C05370=1007.912,298.637,-156.011,2.906,71.013,33.161
C05371=1007.852,298.815,-156.123,3.500,71.107,33.963
C05372=1007.792,298.994,-156.236,4.100,71.198,34.771
C05373=1007.731,299.173,-156.349,4.700,71.282,35.586
C05374=1007.670,299.350,-156.464,5.320,71.368,36.417
C05375=1007.609,299.529,-156.578,5.950,71.452,37.259
C05376=1007.547,299.705,-156.694,6.591,71.533,38.113
C05377=1007.484,299.883,-156.809,7.249,71.615,38.983
C05378=1007.421,300.059,-156.927,7.912,71.693,39.860
C05379=1007.359,300.235,-157.044,8.587,71.769,40.749
C05380=1007.294,300.411,-157.161,9.296,71.851,41.666
C05381=1007.230,300.586,-157.281,9.991,71.920,42.578
C05382=1007.164,300.761,-157.400,10.723,71.997,43.519
C05383=1007.099,300.936,-157.520,11.439,72.060,44.454
C05384=1007.034,301.109,-157.640,12.197,72.133,45.420
C05385=1006.967,301.283,-157.761,12.947,72.195,46.385
C05386=1006.900,301.456,-157.883,13.707,72.254,47.361
C05387=1006.832,301.629,-158.007,14.495,72.315,48.362
C05388=1006.764,301.802,-158.130,15.272,72.365,49.358
C05389=1006.696,301.973,-158.254,16.077,72.419,50.376
C05390=1006.628,302.145,-158.378,16.906,72.473,51.414
C05391=1006.558,302.316,-158.504,17.740,72.521,52.461
C05392=1006.488,302.487,-158.630,18.568,72.561,53.505
C05393=1006.418,302.657,-158.757,19.417,72.600,54.567
C05394=1006.347,302.827,-158.884,20.271,72.636,55.634
C05395=1006.276,302.996,-159.013,21.134,72.666,56.711
C05396=1006.204,303.164,-159.141,22.013,72.694,57.803
C05397=1006.131,303.333,-159.270,22.899,72.718,58.901
C05398=1006.058,303.500,-159.401,23.787,72.735,60.004
C05399=1005.985,303.668,-159.531,24.716,72.757,61.138
C05400=1005.911,303.835,-159.663,25.614,72.764,62.252
C05401=1005.836,304.001,-159.795,26.558,72.775,63.401
C05402=1005.761,304.166,-159.928,27.467,72.773,64.528
C05403=1005.686,304.332,-160.061,28.426,72.776,65.689
C05404=1005.610,304.497,-160.195,29.363,72.767,66.839
C05405=1005.533,304.661,-160.330,30.303,72.753,67.991
C05406=1005.456,304.824,-160.466,31.260,72.738,69.154
C05407=1005.379,304.988,-160.602,32.197,72.712,70.305
C05408=1005.300,305.150,-160.740,33.155,72.686,71.469
C05409=1005.221,305.312,-160.876,34.138,72.658,72.651
C05410=1005.141,305.474,-161.015,35.102,72.622,73.820
C05411=1005.062,305.634,-161.154,36.053,72.578,74.978
C05412=1004.982,305.795,-161.294,37.021,72.531,76.150
C05413=1004.901,305.954,-161.434,37.983,72.478,77.315
C05414=1004.820,306.114,-161.576,38.940,72.419,78.476
C05415=1004.738,306.273,-161.717,39.900,72.356,79.638
C05416=1004.656,306.430,-161.859,40.856,72.287,80.795
C05417=1004.574,306.588,-162.002,41.803,72.212,81.945
C05418=1004.490,306.745,-162.146,42.786,72.137,83.118
C05419=1004.406,306.901,-162.290,43.707,72.048,84.246
C05420=1004.321,307.056,-162.435,44.673,71.960,85.405
C05421=1004.237,307.211,-162.581,45.601,71.862,86.534
C05422=1004.152,307.366,-162.728,46.537,71.762,87.663
C05423=1004.065,307.519,-162.875,47.480,71.659,88.795
C05424=1003.979,307.673,-163.023,48.398,71.548,89.905
C05425=1003.893,307.825,-163.171,49.292,71.430,90.995
C05426=1003.804,307.977,-163.320,50.204,71.310,92.094
C05427=1003.717,308.128,-163.469,51.076,71.182,93.162
C05428=1003.628,308.279,-163.620,51.950,71.050,94.225
C05429=1003.539,308.429,-163.771,52.856,70.919,95.305
C05430=1003.403,308.655,-164.001,54.168,70.704,96.898
C05431=1003.266,308.880,-164.234,55.443,70.477,98.453
C05432=1003.564,308.723,-164.621,36.254,67.418,86.861
C05433=1003.709,308.486,-164.376,34.721,67.533,84.964
C05434=1003.852,308.248,-164.134,33.173,67.628,83.052
C05435=1003.941,308.099,-163.985,32.181,67.673,81.840
C05436=1004.029,307.948,-163.834,31.222,67.719,80.647
C05437=1004.116,307.798,-163.684,30.275,67.761,79.460
C05438=1004.203,307.646,-163.537,29.304,67.790,78.257
C05439=1004.290,307.495,-163.389,28.352,67.817,77.062
C05440=1004.376,307.342,-163.242,27.387,67.834,75.861
C05441=1004.461,307.189,-163.095,26.413,67.842,74.651
C05442=1004.546,307.035,-162.949,25.454,67.846,73.452
C05443=1004.631,306.881,-162.804,24.510,67.847,72.261
C05444=1004.715,306.726,-162.660,23.549,67.834,71.062
C05445=1004.798,306.570,-162.516,22.630,67.826,69.888
C05446=1004.882,306.414,-162.373,21.674,67.798,68.696
C05447=1004.965,306.257,-162.230,20.755,67.774,67.526
C05448=1005.046,306.100,-162.088,19.838,67.741,66.361
C05449=1005.128,305.941,-161.948,18.928,67.702,65.201
C05450=1005.209,305.783,-161.807,18.030,67.658,64.052
C05451=1005.289,305.623,-161.667,17.141,67.609,62.912
C05452=1005.369,305.464,-161.527,16.258,67.553,61.777
C05453=1005.448,305.304,-161.389,15.395,67.495,60.659
C05454=1005.527,305.142,-161.251,14.529,67.427,59.540
C05455=1005.606,304.981,-161.115,13.666,67.351,58.427
C05456=1005.683,304.818,-160.978,12.826,67.274,57.332
C05457=1005.760,304.657,-160.842,12.013,67.199,56.257
C05458=1005.837,304.493,-160.707,11.191,67.112,55.180
C05459=1005.913,304.330,-160.572,10.391,67.024,54.118
C05460=1005.989,304.166,-160.439,9.605,66.933,53.072
C05461=1006.065,304.001,-160.306,8.811,66.828,52.024
C05462=1006.139,303.836,-160.174,8.061,66.733,51.008
C05463=1006.213,303.670,-160.042,7.293,66.621,49.985
C05464=1006.287,303.504,-159.911,6.567,66.518,48.994
C05465=1006.360,303.337,-159.780,5.825,66.398,47.996
C05466=1006.433,303.170,-159.651,5.118,66.286,47.025
C05467=1006.505,303.002,-159.523,4.422,66.168,46.066
C05468=1006.576,302.834,-159.395,3.737,66.047,45.120
C05469=1006.648,302.666,-159.267,3.067,65.924,44.186
C05470=1006.718,302.496,-159.140,2.409,65.798,43.264
C05471=1006.789,302.327,-159.013,1.762,65.669,42.354
C05472=1006.859,302.157,-158.887,1.138,65.542,41.464
C05473=1006.927,301.986,-158.763,0.512,65.406,40.575
C05474=1006.996,301.815,-158.639,-0.106,65.265,39.698
C05475=1007.064,301.644,-158.516,-0.703,65.126,38.837
C05476=1007.132,301.473,-158.392,-1.273,64.994,37.997
C05477=1007.199,301.300,-158.271,-1.850,64.850,37.159
C05478=1007.265,301.128,-158.148,-2.401,64.712,36.342
C05479=1007.332,300.954,-158.027,-2.944,64.570,35.533
C05480=1007.397,300.781,-157.908,-3.488,64.418,34.730
C05481=1007.462,300.607,-157.787,-3.999,64.279,33.952
C05482=1007.527,300.433,-157.669,-4.518,64.126,33.173
C05483=1007.591,300.258,-157.550,-5.009,63.984,32.416
C05484=1007.655,300.083,-157.434,-5.507,63.828,31.659
C05485=1007.718,299.908,-157.317,-5.979,63.682,30.923
C05486=1007.781,299.732,-157.200,-6.442,63.534,30.197
C05487=1007.843,299.556,-157.084,-6.897,63.384,29.481
C05488=1007.905,299.379,-156.969,-7.338,63.236,28.777
C05489=1007.966,299.202,-156.855,-7.774,63.084,28.079
C05490=1008.026,299.024,-156.741,-8.195,62.935,27.397
C05491=1008.087,298.846,-156.628,-8.606,62.787,26.723
C05492=1008.147,298.668,-156.516,-9.014,62.634,26.057
C05493=1008.207,298.490,-156.404,-9.415,62.477,25.400
C05494=1008.265,298.311,-156.293,-9.803,62.325,24.753
C05495=1008.323,298.132,-156.182,-10.171,62.183,24.123
C05496=1008.382,297.953,-156.072,-10.544,62.028,23.494
C05497=1008.439,297.773,-155.962,-10.904,61.877,22.877
C05498=1008.497,297.592,-155.854,-11.264,61.719,22.265
C05499=1008.553,297.411,-155.746,-11.600,61.576,21.669
C05500=1008.609,297.230,-155.639,-11.936,61.426,21.078
C05501=1008.665,297.050,-155.532,-12.269,61.272,20.494
C05502=1008.721,296.868,-155.425,-12.578,61.135,19.926
C05503=1008.775,296.686,-155.319,-12.895,60.982,19.358
C05504=1008.830,296.504,-155.214,-13.200,60.837,18.800
C05505=1008.884,296.322,-155.109,-13.495,60.693,18.254
C05506=1008.937,296.139,-155.006,-13.788,60.546,17.710
C05507=1008.990,295.956,-154.902,-14.070,60.404,17.176
C05508=1009.043,295.773,-154.800,-14.348,60.260,16.650
C05509=1009.095,295.589,-154.698,-14.620,60.116,16.129
C05510=1009.147,295.405,-154.596,-14.882,59.977,15.619
C05511=1009.199,295.221,-154.496,-15.151,59.823,15.108
C05512=1009.249,295.036,-154.395,-15.403,59.684,14.610
C05513=1009.300,294.852,-154.295,-15.643,59.554,14.122
C05514=1009.350,294.666,-154.196,-15.888,59.409,13.636
C05515=1009.400,294.481,-154.097,-16.119,59.279,13.159
C05516=1009.449,294.295,-153.999,-16.352,59.138,12.685
C05517=1009.498,294.110,-153.902,-16.581,58.999,12.216
C05518=1009.548,293.923,-153.805,-16.803,58.861,11.755
C05519=1009.595,293.738,-153.708,-17.013,58.734,11.305
C05520=1009.643,293.550,-153.612,-17.229,58.594,10.853
C05521=1009.690,293.364,-153.517,-17.431,58.467,10.413
C05522=1009.737,293.177,-153.422,-17.636,58.330,9.973
C05523=1009.784,292.989,-153.328,-17.832,58.202,9.541
C05524=1009.830,292.802,-153.235,-18.023,58.075,9.116
///RCONF 0,0,0,0,1,0,0,0,0,0,0,0,0,0,0,0,0,0,0,0,0,0,0,0
C05525=1009.876,292.614,-153.141,-18.212,57.945,8.695
C05526=1009.921,292.425,-153.048,-18.394,57.822,8.281
C05527=1009.966,292.238,-152.957,-18.575,57.694,7.869
C05528=1010.011,292.049,-152.866,-18.754,57.565,7.463
C05529=1010.056,291.860,-152.774,-18.930,57.432,7.061
C05530=1010.099,291.671,-152.683,-19.096,57.314,6.665
C05531=1010.142,291.482,-152.593,-19.257,57.201,6.277
C05532=1010.185,291.292,-152.504,-19.420,57.075,5.890
C05533=1010.228,291.102,-152.414,-19.574,56.964,5.509
C05534=1010.271,290.912,-152.326,-19.731,56.840,5.129
C05535=1010.313,290.723,-152.238,-19.881,56.726,4.757
C05536=1010.354,290.532,-152.151,-20.034,56.600,4.385
C05537=1010.395,290.341,-152.064,-20.177,56.487,4.020
C05538=1010.437,290.151,-151.978,-20.319,56.374,3.660
C05539=1010.478,289.960,-151.892,-20.460,56.255,3.302
C05540=1010.517,289.769,-151.805,-20.593,56.150,2.950
C05541=1010.557,289.578,-151.721,-20.728,56.034,2.598
C05542=1010.597,289.386,-151.637,-20.858,55.925,2.254
C05543=1010.635,289.194,-151.553,-20.985,55.818,1.913
C05544=1010.674,289.002,-151.469,-21.111,55.708,1.575
C05545=1010.713,288.810,-151.386,-21.232,55.603,1.240
C05546=1010.751,288.618,-151.303,-21.353,55.496,0.909
C05547=1010.789,288.426,-151.222,-21.473,55.386,0.580
C05548=1010.827,288.233,-151.140,-21.592,55.273,0.252
C05549=1010.864,288.041,-151.059,-21.704,55.174,-0.068
C05550=1010.900,287.848,-150.977,-21.812,55.079,-0.386
C05551=1010.938,287.654,-150.898,-21.922,54.972,-0.701
C05552=1010.973,287.461,-150.818,-22.027,54.878,-1.014
C05553=1011.009,287.267,-150.739,-22.137,54.764,-1.327
C05554=1011.045,287.074,-150.660,-22.242,54.660,-1.635
C05555=1011.080,286.880,-150.581,-22.340,54.569,-1.937
C05556=1011.114,286.687,-150.503,-22.437,54.478,-2.238
C05557=1011.149,286.492,-150.427,-22.538,54.370,-2.538
C05558=1011.183,286.299,-150.350,-22.634,54.274,-2.835
C05559=1011.250,285.910,-150.196,-22.815,54.098,-3.415
C05560=1011.316,285.521,-150.045,-22.993,53.917,-3.988
C05561=1011.381,285.131,-149.896,-23.164,53.735,-4.549
C05562=1011.445,284.740,-149.749,-23.334,53.544,-5.105
C05563=1011.507,284.349,-149.603,-23.491,53.382,-5.648
C05564=1011.568,283.958,-149.459,-23.644,53.215,-6.185
C05565=1011.627,283.566,-149.316,-23.794,53.047,-6.716
C05566=1011.687,283.174,-149.176,-23.942,52.870,-7.241
C05567=1011.744,282.781,-149.037,-24.081,52.710,-7.756
C05568=1011.800,282.387,-148.900,-24.215,52.554,-8.265
C05569=1011.855,281.993,-148.764,-24.347,52.396,-8.768
C05570=1011.909,281.600,-148.630,-24.474,52.242,-9.263
C05571=1011.962,281.204,-148.499,-24.599,52.079,-9.755
C05572=1012.013,280.810,-148.367,-24.716,51.938,-10.234
C05573=1012.063,280.414,-148.239,-24.832,51.789,-10.711
C05574=1012.113,280.018,-148.110,-24.944,51.641,-11.182
C05575=1012.161,279.622,-147.985,-25.053,51.494,-11.648
C05576=1012.208,279.226,-147.861,-25.157,51.361,-12.105
C05577=1012.254,278.830,-147.738,-25.259,51.217,-12.557
C05578=1012.298,278.432,-147.616,-25.356,51.098,-13.003
C05579=1012.342,278.035,-147.497,-25.452,50.965,-13.448
C05580=1012.385,277.637,-147.379,-25.548,50.816,-13.891
C05581=1012.426,277.238,-147.262,-25.636,50.709,-14.325
C05582=1012.467,276.841,-147.147,-25.726,50.572,-14.760
C05583=1012.506,276.442,-147.034,-25.811,50.451,-15.189
C05584=1012.544,276.043,-146.922,-25.896,50.325,-15.616
C05585=1012.581,275.644,-146.812,-25.978,50.199,-16.040
C05586=1012.618,275.245,-146.703,-26.058,50.077,-16.460
C05587=1012.653,274.845,-146.596,-26.135,49.965,-16.875
C05588=1012.687,274.446,-146.490,-26.210,49.849,-17.287
C05589=1012.720,274.045,-146.386,-26.286,49.721,-17.699
C05590=1012.752,273.644,-146.283,-26.357,49.609,-18.105
C05591=1012.783,273.244,-146.181,-26.426,49.502,-18.508
C05592=1012.812,272.843,-146.081,-26.494,49.400,-18.906
C05593=1012.843,272.442,-145.983,-26.562,49.264,-19.308
C05594=1012.870,272.041,-145.886,-26.626,49.168,-19.700
C05595=1012.896,271.640,-145.790,-26.690,49.055,-20.094
C05596=1012.922,271.238,-145.696,-26.752,48.946,-20.485
C05597=1012.947,270.836,-145.604,-26.812,48.854,-20.871
C05598=1012.971,270.434,-145.513,-26.871,48.735,-21.260
C05599=1012.993,270.032,-145.422,-26.928,48.656,-21.639
C05600=1013.016,269.630,-145.335,-26.985,48.544,-22.024
C05601=1013.036,269.228,-145.247,-27.040,48.454,-22.404
C05602=1013.057,268.825,-145.163,-27.094,48.326,-22.787
C05603=1013.076,268.422,-145.078,-27.146,48.239,-23.161
C05604=1013.093,268.019,-144.996,-27.198,48.146,-23.537
C05605=1013.110,267.615,-144.915,-27.248,48.034,-23.913
C05606=1013.126,267.212,-144.835,-27.297,47.964,-24.279
C05607=1013.141,266.808,-144.757,-27.345,47.858,-24.651
C05608=1013.155,266.405,-144.680,-27.392,47.768,-25.018
C05609=1013.168,266.002,-144.605,-27.438,47.689,-25.383
C05610=1013.180,265.597,-144.530,-27.483,47.598,-25.747
C05611=1013.191,265.193,-144.458,-27.527,47.493,-26.113
C05612=1013.202,264.789,-144.388,-27.569,47.395,-26.476
C05613=1013.210,264.385,-144.317,-27.612,47.337,-26.831
C05614=1013.219,263.981,-144.250,-27.652,47.223,-27.196
C05615=1013.226,263.576,-144.182,-27.692,47.141,-27.552
C05616=1013.232,263.171,-144.116,-27.732,47.074,-27.905
C05617=1013.236,262.903,-144.075,-27.757,47.002,-28.143
C05618=1013.239,262.635,-144.033,-27.782,46.948,-28.378
C05619=1013.242,262.367,-143.990,-27.808,46.911,-28.609
C05620=1013.244,262.099,-143.950,-27.832,46.851,-28.843
C05621=1013.246,261.825,-143.908,-27.857,46.794,-29.081
C05622=1013.247,261.551,-143.868,-27.882,46.748,-29.317
C05623=1013.250,261.146,-143.811,-27.915,46.638,-29.673
C05624=1013.250,260.741,-143.753,-27.950,46.568,-30.019
C05625=1013.249,260.336,-143.697,-27.984,46.495,-30.366
C05626=1013.249,259.930,-143.643,-28.016,46.399,-30.715
C05627=1013.246,259.525,-143.589,-28.050,46.343,-31.056
C05628=1013.233,258.298,-143.437,-28.144,46.129,-32.080
C05629=1013.230,258.053,-143.408,-28.143,46.117,-32.083
C05630=1013.227,257.808,-143.379,-28.142,46.105,-32.086
C05631=1013.223,257.563,-143.350,-28.141,46.093,-32.089
C05632=1013.220,257.318,-143.321,-28.140,46.083,-32.091
C05633=1013.217,257.072,-143.292,-28.139,46.072,-32.095
C05634=1013.214,256.827,-143.263,-28.138,46.062,-32.097
C05635=1013.211,256.583,-143.234,-28.137,46.052,-32.100
C05636=1013.208,256.337,-143.205,-28.137,46.043,-32.103
C05637=1013.204,256.092,-143.176,-28.136,46.034,-32.106
C05638=1013.201,255.847,-143.147,-28.135,46.025,-32.108
C05639=1013.198,255.602,-143.118,-28.134,46.014,-32.111
C05640=1013.195,255.358,-143.089,-28.133,46.003,-32.114
C05641=1013.192,255.112,-143.061,-28.132,45.991,-32.117
C05642=1013.189,254.867,-143.032,-28.131,45.979,-32.120
C05643=1013.186,254.622,-143.003,-28.131,45.969,-32.122
C05644=1013.183,254.377,-142.973,-28.130,45.958,-32.126
C05645=1013.179,254.132,-142.944,-28.129,45.948,-32.128
C05646=1013.176,253.886,-142.916,-28.128,45.938,-32.131
C05647=1013.173,253.641,-142.887,-28.127,45.929,-32.134
C05648=1013.170,253.396,-142.858,-28.127,45.919,-32.136
C05649=1013.167,253.151,-142.829,-28.126,45.910,-32.139
C05650=1013.163,252.906,-142.800,-28.125,45.900,-32.142
C05651=1013.160,252.661,-142.772,-28.124,45.888,-32.144
C05652=1013.158,252.416,-142.743,-28.123,45.876,-32.147
C05653=1013.155,252.171,-142.714,-28.122,45.865,-32.151
C05654=1013.152,251.925,-142.686,-28.121,45.853,-32.154
C05655=1013.148,251.680,-142.657,-28.120,45.843,-32.156
C05656=1013.146,251.435,-142.627,-28.119,45.833,-32.159
C05657=1013.142,251.190,-142.599,-28.119,45.823,-32.163
C05658=1013.139,250.945,-142.570,-28.118,45.813,-32.165
C05659=1013.136,250.700,-142.542,-28.117,45.804,-32.167
C05660=1013.134,250.454,-142.513,-28.116,45.795,-32.170
C05661=1013.130,250.209,-142.484,-28.115,45.783,-32.173
C05662=1013.127,249.964,-142.456,-28.114,45.772,-32.176
C05663=1013.124,249.719,-142.427,-28.113,45.760,-32.179
C05664=1013.121,249.473,-142.398,-28.112,45.748,-32.182
C05665=1013.119,249.229,-142.370,-28.111,45.738,-32.184
C05666=1013.116,248.983,-142.342,-28.111,45.727,-32.188
C05667=1013.112,248.738,-142.313,-28.110,45.717,-32.190
C05668=1013.110,248.492,-142.284,-28.109,45.707,-32.193
C05669=1013.106,248.247,-142.255,-28.108,45.697,-32.195
C05670=1013.104,248.002,-142.227,-28.107,45.688,-32.198
C05671=1013.100,247.757,-142.199,-28.107,45.678,-32.201
C05672=1013.098,247.511,-142.170,-28.106,45.667,-32.204
C05673=1013.095,247.266,-142.141,-28.104,45.654,-32.207
C05674=1013.092,247.022,-142.113,-28.103,45.642,-32.210
C05675=1013.089,246.776,-142.085,-28.103,45.631,-32.213
C05676=1013.086,246.531,-142.055,-28.102,45.620,-32.215
C05677=1013.083,246.285,-142.027,-28.101,45.609,-32.219
C05678=1013.080,246.041,-141.999,-28.100,45.599,-32.221
C05679=1013.077,245.795,-141.971,-28.099,45.589,-32.223
C05680=1013.075,245.549,-141.942,-28.098,45.580,-32.226
C05681=1013.071,245.304,-141.913,-28.097,45.570,-32.229
C05682=1013.069,245.059,-141.885,-28.097,45.561,-32.232
C05683=1013.066,244.814,-141.857,-28.095,45.548,-32.234
C05684=1013.063,244.569,-141.827,-28.094,45.536,-32.237
C05685=1013.061,244.324,-141.800,-28.093,45.524,-32.240
C05686=1013.057,244.078,-141.772,-28.092,45.513,-32.243
C05687=1013.054,243.832,-141.743,-28.092,45.503,-32.246
C05688=1013.053,243.587,-141.715,-28.091,45.492,-32.249
C05689=1013.049,243.342,-141.686,-28.090,45.482,-32.252
C05690=1013.046,243.097,-141.658,-28.089,45.472,-32.254
C05691=1013.044,242.852,-141.630,-28.088,45.461,-32.257
C05692=1013.041,242.606,-141.601,-28.087,45.452,-32.260
C05693=1013.038,242.361,-141.572,-28.086,45.440,-32.263
C05694=1013.035,242.116,-141.545,-28.085,45.429,-32.266
C05695=1013.032,241.870,-141.516,-28.084,45.417,-32.269
C05696=1013.030,241.625,-141.488,-28.083,45.405,-32.272
C05697=1013.027,241.380,-141.460,-28.082,45.394,-32.274
C05698=1013.024,241.134,-141.432,-28.081,45.383,-32.277
C05699=1013.022,240.889,-141.404,-28.080,45.372,-32.279
C05700=1013.019,240.643,-141.375,-28.079,45.361,-32.283
C05701=1013.016,240.398,-141.347,-28.079,45.351,-32.285
C05702=1013.014,240.153,-141.319,-28.078,45.342,-32.288
C05703=1013.010,239.907,-141.291,-28.077,45.333,-32.289
C05704=1013.008,239.662,-141.263,-28.076,45.321,-32.292
C05705=1013.006,239.416,-141.234,-28.075,45.308,-32.297
C05706=1013.003,239.171,-141.207,-28.074,45.297,-32.300
C05707=1013.000,238.926,-141.179,-28.073,45.286,-32.301
C05708=1012.997,238.681,-141.151,-28.072,45.274,-32.305
C05709=1012.995,238.435,-141.122,-28.071,45.262,-32.308
C05710=1012.992,238.189,-141.094,-28.070,45.252,-32.310
C05711=1012.989,237.945,-141.066,-28.069,45.242,-32.312
C05712=1012.986,237.699,-141.038,-28.068,45.232,-32.315
C05713=1012.985,237.454,-141.009,-28.067,45.223,-32.318
C05714=1012.981,237.208,-140.981,-28.067,45.213,-32.320
C05715=1012.979,236.963,-140.953,-28.065,45.199,-32.324
C05716=1012.976,236.718,-140.925,-28.064,45.187,-32.327
C05717=1012.974,236.473,-140.897,-28.063,45.176,-32.330
C05718=1012.971,236.226,-140.869,-28.062,45.165,-32.332
C05719=1012.969,235.981,-140.842,-28.061,45.153,-32.335
C05720=1012.966,235.736,-140.813,-28.060,45.141,-32.338
C05721=1012.964,235.491,-140.785,-28.059,45.131,-32.340
C05722=1012.961,235.245,-140.757,-28.058,45.121,-32.343
C05723=1012.958,234.999,-140.730,-28.058,45.111,-32.345
C05724=1012.955,234.754,-140.702,-28.057,45.101,-32.348
C05725=1012.954,234.509,-140.673,-28.056,45.090,-32.351
C05726=1012.950,234.263,-140.645,-28.055,45.077,-32.354
C05727=1012.948,234.018,-140.618,-28.054,45.066,-32.357
C05728=1012.946,233.773,-140.590,-28.053,45.054,-32.360
C05729=1012.943,233.527,-140.561,-28.052,45.042,-32.363
C05730=1012.941,233.282,-140.534,-28.051,45.030,-32.366
C05731=1012.938,233.036,-140.506,-28.049,45.019,-32.368
C05732=1012.936,232.791,-140.478,-28.049,45.009,-32.370
C05733=1012.933,232.545,-140.450,-28.048,44.998,-32.374
C05734=1012.931,232.299,-140.423,-28.047,44.988,-32.377
C05735=1012.928,232.054,-140.394,-28.046,44.978,-32.379
C05736=1012.925,231.809,-140.367,-28.045,44.966,-32.382
C05737=1012.924,231.563,-140.339,-28.044,44.955,-32.385
C05738=1012.921,231.317,-140.311,-28.043,44.942,-32.388
C05739=1012.919,231.072,-140.284,-28.042,44.930,-32.391
C05740=1012.916,230.827,-140.256,-28.041,44.918,-32.394
C05741=1012.914,230.580,-140.228,-28.039,44.908,-32.396
C05742=1012.911,230.336,-140.200,-28.039,44.897,-32.399
C05743=1012.909,230.089,-140.172,-28.038,44.886,-32.401
C05744=1012.907,229.844,-140.144,-28.037,44.876,-32.404
C05745=1012.904,229.599,-140.116,-28.036,44.866,-32.406
C05746=1012.902,229.353,-140.089,-28.035,44.855,-32.408
C05747=1012.899,229.108,-140.061,-28.034,44.843,-32.413
C05748=1012.898,228.862,-140.033,-28.033,44.830,-32.415
C05749=1012.895,228.616,-140.006,-28.032,44.818,-32.419
C05750=1012.892,228.371,-139.978,-28.030,44.806,-32.421
C05751=1012.890,228.126,-139.951,-28.029,44.794,-32.424
C05752=1012.888,227.880,-139.922,-28.028,44.783,-32.426
C05753=1012.885,227.634,-139.895,-28.027,44.772,-32.430
C05754=1012.883,227.389,-139.867,-28.026,44.762,-32.432
C05755=1012.880,227.143,-139.840,-28.025,44.751,-32.434
C05756=1012.879,226.897,-139.812,-28.025,44.740,-32.438
C05757=1012.876,226.652,-139.784,-28.024,44.730,-32.440
C05758=1012.873,226.406,-139.757,-28.022,44.718,-32.443
C05759=1012.872,226.161,-139.729,-28.021,44.706,-32.446
C05760=1012.869,225.915,-139.701,-28.020,44.693,-32.448
C05761=1012.867,225.670,-139.674,-28.019,44.681,-32.451
C05762=1012.864,225.424,-139.647,-28.018,44.670,-32.454
C05763=1012.863,225.179,-139.619,-28.017,44.658,-32.458
C05764=1012.860,224.933,-139.591,-28.016,44.647,-32.459
C05765=1012.858,224.687,-139.564,-28.015,44.636,-32.463
C05766=1012.856,224.442,-139.536,-28.014,44.626,-32.466
C05767=1012.854,224.196,-139.509,-28.013,44.616,-32.468
C05768=1012.851,223.951,-139.481,-28.012,44.604,-32.471
C05769=1012.849,223.704,-139.454,-28.011,44.592,-32.474
C05770=1012.847,223.459,-139.426,-28.010,44.579,-32.476
C05771=1012.845,223.214,-139.399,-28.009,44.567,-32.479
C05772=1012.842,222.968,-139.371,-28.008,44.555,-32.482
C05773=1012.840,222.722,-139.343,-28.007,44.544,-32.486
C05774=1012.838,222.476,-139.316,-28.006,44.532,-32.489
C05775=1012.836,222.231,-139.289,-28.005,44.521,-32.491
C05776=1012.833,221.986,-139.261,-28.004,44.510,-32.494
C05777=1012.831,221.739,-139.233,-28.003,44.500,-32.497
C05778=1012.829,221.494,-139.206,-28.002,44.489,-32.499
C05779=1012.827,221.248,-139.179,-28.001,44.477,-32.502
C05780=1012.825,221.002,-139.151,-28.000,44.465,-32.505
C05781=1012.823,220.757,-139.124,-27.998,44.454,-32.507
C05782=1012.821,220.511,-139.097,-27.998,44.444,-32.510
C05783=1012.819,220.266,-139.070,-27.997,44.432,-32.514
C05784=1012.817,220.017,-139.042,-27.995,44.420,-32.517
C05785=1012.815,219.757,-139.013,-27.994,44.407,-32.521
C05786=1012.812,219.484,-138.983,-27.993,44.394,-32.525
C05787=1012.810,219.202,-138.951,-27.992,44.381,-32.528
C05788=1012.807,218.907,-138.918,-27.991,44.367,-32.531
C05789=1012.805,218.603,-138.884,-27.989,44.353,-32.532
C05790=1012.802,218.308,-138.851,-27.988,44.339,-32.536
C05791=1012.800,218.014,-138.819,-27.987,44.325,-32.538
C05792=1012.797,217.724,-138.787,-27.985,44.312,-32.539
C05793=1012.795,217.444,-138.756,-27.984,44.298,-32.543
C05794=1012.793,217.180,-138.726,-27.983,44.286,-32.546
C05795=1012.790,216.920,-138.698,-27.982,44.273,-32.550
C05796=1012.788,216.665,-138.669,-27.981,44.260,-32.555
C05797=1012.786,216.417,-138.641,-27.980,44.249,-32.558
C05798=1012.784,216.172,-138.614,-27.979,44.237,-32.561
C05799=1012.782,215.926,-138.587,-27.977,44.224,-32.564
C05800=1012.780,215.680,-138.560,-27.976,44.213,-32.566
C05801=1012.779,215.436,-138.533,-27.975,44.201,-32.569
C05802=1012.776,215.190,-138.506,-27.974,44.190,-32.572
C05803=1012.774,214.945,-138.479,-27.973,44.178,-32.575
C05804=1012.773,214.700,-138.452,-27.972,44.166,-32.578
C05805=1012.771,214.455,-138.425,-27.971,44.155,-32.580
C05806=1012.768,214.210,-138.397,-27.970,44.143,-32.583
C05807=1012.767,213.965,-138.371,-27.969,44.131,-32.586
C05808=1012.765,213.721,-138.343,-27.968,44.119,-32.589
C05809=1012.763,213.478,-138.317,-27.967,44.107,-32.592
C05810=1012.761,213.233,-138.290,-27.965,44.096,-32.594
C05811=1012.759,212.989,-138.263,-27.964,44.085,-32.597
C05812=1012.757,212.746,-138.236,-27.963,44.072,-32.600
C05813=1012.756,212.502,-138.209,-27.962,44.060,-32.603
C05814=1012.754,212.259,-138.183,-27.961,44.048,-32.606
C05815=1012.752,212.017,-138.155,-27.960,44.037,-32.610
C05816=1012.749,211.774,-138.129,-27.959,44.026,-32.611
C05817=1012.748,211.530,-138.102,-27.958,44.014,-32.615
C05818=1012.746,211.287,-138.075,-27.957,44.002,-32.618
C05819=1012.744,211.045,-138.049,-27.955,43.990,-32.620
C05820=1012.742,210.802,-138.022,-27.954,43.978,-32.624
C05821=1012.741,210.560,-137.995,-27.953,43.966,-32.627
C05822=1012.738,210.317,-137.969,-27.952,43.954,-32.630
C05823=1012.737,210.075,-137.942,-27.951,43.942,-32.633
C05824=1012.735,209.833,-137.916,-27.950,43.930,-32.636
C05825=1012.733,209.590,-137.889,-27.949,43.918,-32.639
C05826=1012.732,209.347,-137.862,-27.948,43.907,-32.641
C05827=1012.730,209.106,-137.835,-27.947,43.896,-32.644
C05828=1012.728,208.863,-137.809,-27.946,43.883,-32.649
C05829=1012.727,208.621,-137.782,-27.944,43.871,-32.650
C05830=1012.725,208.378,-137.756,-27.943,43.859,-32.653
C05831=1012.723,208.136,-137.729,-27.942,43.848,-32.656
C05832=1012.721,207.893,-137.702,-27.941,43.836,-32.659
C05833=1012.720,207.651,-137.676,-27.940,43.824,-32.663
C05834=1012.717,207.408,-137.649,-27.939,43.812,-32.666
C05835=1012.716,207.166,-137.623,-27.938,43.801,-32.669
C05836=1012.714,206.923,-137.597,-27.937,43.788,-32.672
C05837=1012.713,206.679,-137.570,-27.936,43.776,-32.675
C05838=1012.711,206.437,-137.543,-27.935,43.764,-32.678
C05839=1012.709,206.194,-137.517,-27.933,43.753,-32.681
C05840=1012.708,205.950,-137.490,-27.932,43.741,-32.682
C05841=1012.706,205.707,-137.463,-27.931,43.729,-32.686
C05842=1012.704,205.464,-137.437,-27.930,43.717,-32.689
C05843=1012.703,205.220,-137.411,-27.929,43.705,-32.692
C05844=1012.701,204.976,-137.383,-27.928,43.693,-32.695
C05845=1012.699,204.732,-137.357,-27.927,43.681,-32.698
C05846=1012.697,204.488,-137.330,-27.925,43.669,-32.701
C05847=1012.696,204.244,-137.304,-27.924,43.657,-32.704
C05848=1012.694,203.999,-137.277,-27.923,43.644,-32.706
C05849=1012.692,203.754,-137.251,-27.922,43.632,-32.710
C05850=1012.691,203.510,-137.224,-27.921,43.620,-32.712
C05851=1012.689,203.262,-137.197,-27.920,43.608,-32.715
C05852=1012.686,202.023,-137.060,-27.878,43.638,-32.166
C05853=1012.687,201.804,-137.037,-27.877,43.626,-32.169
C05854=1012.687,201.599,-137.014,-27.876,43.616,-32.172
C05855=1012.689,201.183,-136.969,-27.874,43.594,-32.177
C05856=1012.689,200.965,-136.946,-27.873,43.582,-32.181
C05857=1012.689,200.743,-136.921,-27.872,43.571,-32.184
C05858=1012.690,200.504,-136.896,-27.871,43.558,-32.188
C05859=1012.690,200.249,-136.868,-27.870,43.545,-32.191
C05860=1012.691,199.995,-136.841,-27.869,43.532,-32.196
C05861=1012.691,199.754,-136.815,-27.868,43.519,-32.200
C05862=1012.692,199.521,-136.789,-27.867,43.507,-32.203
C05863=1012.692,199.292,-136.765,-27.866,43.495,-32.206
C05864=1012.693,199.050,-136.738,-27.865,43.483,-32.211
C05865=1012.694,198.660,-136.697,-27.863,43.462,-32.216
C05866=1012.695,198.269,-136.654,-27.861,43.442,-32.223
C05867=1012.696,198.022,-136.627,-27.860,43.429,-32.227
C05868=1012.696,197.786,-136.601,-27.859,43.416,-32.230
C05869=1012.697,197.550,-136.576,-27.858,43.403,-32.234
C05870=1012.697,197.314,-136.550,-27.857,43.390,-32.238
C05871=1012.698,197.078,-136.525,-27.856,43.378,-32.242
C05872=1012.699,196.842,-136.500,-27.855,43.366,-32.245
C05873=1012.699,196.606,-136.474,-27.854,43.355,-32.248
C05874=1012.700,196.370,-136.449,-27.853,43.342,-32.253
C05875=1012.700,196.134,-136.423,-27.852,43.332,-32.256
C05876=1012.701,195.899,-136.398,-27.851,43.320,-32.259
C05877=1012.701,195.663,-136.373,-27.850,43.307,-32.263
C05878=1012.703,195.427,-136.348,-27.849,43.294,-32.268
C05879=1012.703,195.191,-136.323,-27.848,43.282,-32.271
C05880=1012.704,194.955,-136.297,-27.847,43.270,-32.275
C05881=1012.704,194.719,-136.272,-27.846,43.258,-32.279
C05882=1012.704,194.483,-136.246,-27.845,43.246,-32.282
C05883=1012.706,194.248,-136.221,-27.844,43.234,-32.285
C05884=1012.706,194.012,-136.196,-27.843,43.222,-32.289
C05885=1012.707,193.776,-136.170,-27.842,43.212,-32.293
C05886=1012.708,193.539,-136.144,-27.841,43.200,-32.296
C05887=1012.709,193.304,-136.119,-27.840,43.187,-32.301
C05888=1012.709,193.068,-136.094,-27.838,43.174,-32.303
C05889=1012.710,192.832,-136.068,-27.837,43.162,-32.308
C05890=1012.710,192.596,-136.043,-27.836,43.150,-32.311
C05891=1012.711,192.361,-136.018,-27.835,43.137,-32.316
C05892=1012.712,192.124,-135.993,-27.834,43.126,-32.319
C05893=1012.713,191.888,-135.968,-27.833,43.114,-32.322
C05894=1012.713,191.652,-135.942,-27.832,43.103,-32.326
C05895=1012.714,191.417,-135.917,-27.831,43.091,-32.330
C05896=1012.715,191.181,-135.892,-27.830,43.080,-32.334
C05897=1012.715,190.945,-135.866,-27.829,43.068,-32.337
C05898=1012.716,190.709,-135.841,-27.828,43.055,-32.341
C05899=1012.717,190.474,-135.816,-27.827,43.042,-32.346
C05900=1012.717,190.237,-135.791,-27.826,43.031,-32.349
C05901=1012.718,190.001,-135.765,-27.825,43.019,-32.352
C05902=1012.719,189.766,-135.740,-27.824,43.007,-32.356
C05903=1012.719,189.530,-135.715,-27.823,42.996,-32.359
C05904=1012.720,189.294,-135.689,-27.822,42.984,-32.363
C05905=1012.721,189.059,-135.664,-27.821,42.973,-32.367
C05906=1012.722,188.822,-135.639,-27.820,42.962,-32.371
C05907=1012.722,188.586,-135.614,-27.819,42.949,-32.375
C05908=1012.723,188.351,-135.589,-27.818,42.937,-32.378
C05909=1012.724,188.115,-135.563,-27.817,42.925,-32.383
C05910=1012.725,187.880,-135.538,-27.816,42.913,-32.386
C05911=1012.725,187.644,-135.514,-27.815,42.901,-32.389
C05912=1012.725,187.408,-135.489,-27.814,42.888,-32.394
C05913=1012.726,187.172,-135.464,-27.813,42.877,-32.398
C05914=1012.727,186.936,-135.438,-27.812,42.866,-32.402
C05915=1012.727,186.700,-135.413,-27.811,42.855,-32.404
C05916=1012.729,186.465,-135.388,-27.810,42.845,-32.408
C05917=1012.729,186.229,-135.363,-27.809,42.832,-32.412
C05918=1012.730,185.993,-135.338,-27.808,42.820,-32.416
C05919=1012.731,185.757,-135.312,-27.807,42.808,-32.421
C05920=1012.732,185.521,-135.288,-27.806,42.796,-32.424
C05921=1012.733,185.286,-135.263,-27.805,42.784,-32.427
C05922=1012.733,185.050,-135.237,-27.804,42.773,-32.431
C05923=1012.734,184.814,-135.212,-27.803,42.761,-32.434
C05924=1012.735,184.578,-135.187,-27.802,42.750,-32.438
C05925=1012.736,184.342,-135.162,-27.801,42.739,-32.442
C05926=1012.737,184.107,-135.137,-27.800,42.728,-32.446
C05927=1012.738,183.871,-135.112,-27.799,42.715,-32.450
C05928=1012.738,183.635,-135.087,-27.798,42.703,-32.454
C05929=1012.739,183.399,-135.062,-27.797,42.691,-32.457
C05930=1012.739,183.164,-135.037,-27.796,42.680,-32.462
C05931=1012.741,182.928,-135.013,-27.795,42.668,-32.466
C05932=1012.741,182.692,-134.987,-27.794,42.657,-32.470
C05933=1012.742,182.457,-134.962,-27.793,42.645,-32.473
C05934=1012.743,182.221,-134.937,-27.792,42.634,-32.477
C05935=1012.744,181.985,-134.912,-27.791,42.623,-32.481
C05936=1012.744,181.749,-134.887,-27.790,42.612,-32.485
C05937=1012.746,181.514,-134.862,-27.789,42.601,-32.488
C05938=1012.746,181.277,-134.837,-27.788,42.589,-32.491
C05939=1012.747,181.042,-134.812,-27.787,42.576,-32.496
C05940=1012.748,180.806,-134.786,-27.786,42.564,-32.500
C05941=1012.749,180.570,-134.763,-27.785,42.553,-32.503
C05942=1012.749,180.334,-134.737,-27.784,42.542,-32.507
C05943=1012.750,180.099,-134.712,-27.783,42.531,-32.511
C05944=1012.751,179.862,-134.687,-27.782,42.520,-32.515
C05945=1012.752,179.627,-134.662,-27.781,42.509,-32.519
C05946=1012.753,179.392,-134.637,-27.780,42.498,-32.523
C05947=1012.754,179.155,-134.612,-27.779,42.486,-32.526
C05948=1012.755,178.920,-134.587,-27.778,42.474,-32.531
C05949=1012.755,178.684,-134.562,-27.777,42.463,-32.535
C05950=1012.756,178.448,-134.538,-27.776,42.451,-32.538
C05951=1012.757,178.213,-134.513,-27.775,42.440,-32.542
C05952=1012.758,177.977,-134.488,-27.774,42.428,-32.545
C05953=1012.759,177.741,-134.463,-27.773,42.417,-32.549
C05954=1012.760,177.506,-134.438,-27.772,42.406,-32.553
C05955=1012.761,177.270,-134.413,-27.771,42.396,-32.556
C05956=1012.761,177.035,-134.389,-27.770,42.384,-32.561
C05957=1012.762,176.799,-134.363,-27.769,42.373,-32.565
C05958=1012.763,176.563,-134.339,-27.768,42.361,-32.568
C05959=1012.764,176.327,-134.314,-27.767,42.349,-32.573
C05960=1012.765,176.092,-134.289,-27.766,42.337,-32.577
C05961=1012.766,175.856,-134.264,-27.765,42.326,-32.581
C05962=1012.766,175.621,-134.240,-27.764,42.315,-32.585
C05963=1012.768,175.385,-134.215,-27.763,42.305,-32.587
C05964=1012.768,175.149,-134.190,-27.762,42.294,-32.591
C05965=1012.770,174.913,-134.165,-27.761,42.283,-32.595
C05966=1012.771,174.678,-134.140,-27.760,42.272,-32.599
C05967=1012.770,174.442,-134.115,-27.759,42.261,-32.602
C05968=1012.772,174.206,-134.091,-27.758,42.249,-32.608
C05969=1012.773,173.971,-134.066,-27.757,42.237,-32.611
C05970=1012.774,173.735,-134.042,-27.756,42.226,-32.615
C05971=1012.775,173.499,-134.016,-27.755,42.215,-32.619
C05972=1012.775,173.263,-133.992,-27.754,42.204,-32.623
C05973=1012.776,173.028,-133.967,-27.753,42.193,-32.627
C05974=1012.777,172.793,-133.942,-27.752,42.183,-32.630
C05975=1012.778,172.556,-133.917,-27.751,42.172,-32.634
C05976=1012.779,172.321,-133.892,-27.750,42.161,-32.638
C05977=1012.780,172.086,-133.868,-27.749,42.149,-32.642
C05978=1012.781,171.850,-133.843,-27.748,42.138,-32.646
C05979=1012.782,171.614,-133.819,-27.747,42.127,-32.650
C05980=1012.783,171.378,-133.794,-27.746,42.115,-32.654
C05981=1012.784,171.143,-133.770,-27.745,42.104,-32.658
C05982=1012.785,170.908,-133.745,-27.744,42.093,-32.662
C05983=1012.786,170.672,-133.720,-27.743,42.084,-32.665
C05984=1012.787,170.436,-133.695,-27.742,42.073,-32.669
C05985=1012.787,170.201,-133.670,-27.741,42.062,-32.673
C05986=1012.788,169.965,-133.646,-27.740,42.051,-32.677
C05987=1012.789,169.730,-133.621,-27.739,42.040,-32.680
C05988=1012.790,169.494,-133.597,-27.738,42.028,-32.685
C05989=1012.791,169.259,-133.572,-27.737,42.017,-32.689
C05990=1012.792,169.023,-133.548,-27.736,42.006,-32.693
C05991=1012.793,168.788,-133.523,-27.735,41.996,-32.696
C05992=1012.793,168.551,-133.498,-27.734,41.985,-32.700
C05993=1012.795,168.316,-133.473,-27.733,41.974,-32.704
C05994=1012.796,168.080,-133.449,-27.732,41.964,-32.709
C05995=1012.796,167.845,-133.424,-27.731,41.954,-32.711
C05996=1012.798,167.609,-133.400,-27.730,41.941,-32.716
C05997=1012.799,167.374,-133.375,-27.729,41.930,-32.720
C05998=1012.800,167.138,-133.351,-27.728,41.919,-32.724
C05999=1012.800,166.903,-133.326,-27.727,41.908,-32.728
C06000=1012.802,166.668,-133.302,-27.726,41.897,-32.732
C06001=1012.803,166.432,-133.277,-27.725,41.887,-32.736
C06002=1012.804,166.197,-133.253,-27.724,41.876,-32.739
C06003=1012.804,165.961,-133.227,-27.723,41.866,-32.743
C06004=1012.805,165.725,-133.203,-27.722,41.855,-32.747
C06005=1012.806,165.490,-133.179,-27.722,41.846,-32.750
C06006=1012.807,165.254,-133.154,-27.721,41.835,-32.754
C06007=1012.808,165.019,-133.129,-27.720,41.824,-32.758
C06008=1012.809,164.716,-133.098,-27.718,41.810,-32.764
C06009=1012.810,164.398,-133.065,-27.717,41.797,-32.768
C06010=1012.811,164.124,-133.036,-27.716,41.784,-32.773
C06011=1012.813,163.789,-133.001,-27.715,41.768,-32.779
C06012=1012.814,163.568,-132.978,-27.714,41.759,-32.782
C06013=1012.815,163.332,-132.954,-27.713,41.748,-32.786
C06014=1012.816,163.068,-132.926,-27.712,41.735,-32.791
C06015=1012.817,162.775,-132.896,-27.710,41.723,-32.796
C06016=1012.819,162.467,-132.864,-27.709,41.708,-32.802
C06017=1012.820,162.176,-132.833,-27.708,41.696,-32.806
C06018=1012.821,161.869,-132.802,-27.707,41.682,-32.810
C06019=1012.822,161.565,-132.771,-27.705,41.668,-32.816
C06020=1012.824,161.273,-132.741,-27.704,41.655,-32.821
C06021=1012.825,160.995,-132.711,-27.703,41.642,-32.825
C06022=1012.826,160.733,-132.684,-27.702,41.629,-32.830
C06023=1012.827,160.484,-132.658,-27.701,41.618,-32.835
C06024=1012.828,160.243,-132.633,-27.700,41.607,-32.839
C06025=1012.829,160.009,-132.609,-27.699,41.596,-32.843
C06026=1012.832,159.778,-132.587,-27.692,41.528,-32.862
C06027=1012.836,159.545,-132.567,-27.680,41.401,-32.900
C06028=1012.841,159.311,-132.546,-27.667,41.274,-32.937
C06029=1012.845,159.074,-132.526,-27.655,41.145,-32.973
C06030=1012.850,158.838,-132.506,-27.642,41.017,-33.010
C06031=1012.854,158.603,-132.485,-27.629,40.889,-33.048
C06032=1012.858,158.368,-132.465,-27.616,40.761,-33.085
C06033=1012.863,158.132,-132.444,-27.604,40.633,-33.125
C06034=1012.867,157.896,-132.422,-27.591,40.506,-33.162
C06035=1012.872,157.659,-132.402,-27.577,40.376,-33.201
C06036=1012.876,157.421,-132.382,-27.564,40.248,-33.239
C06037=1012.881,157.183,-132.361,-27.551,40.120,-33.278
C06038=1012.886,156.944,-132.340,-27.537,39.989,-33.318
C06039=1012.890,156.704,-132.319,-27.524,39.861,-33.358
C06040=1012.895,156.465,-132.298,-27.511,39.732,-33.397
C06041=1012.901,156.138,-132.270,-27.492,39.556,-33.451
C06042=1012.909,155.748,-132.236,-27.469,39.345,-33.518
C06043=1012.913,155.508,-132.215,-27.455,39.216,-33.558
C06044=1012.918,155.269,-132.193,-27.442,39.089,-33.599
C06045=1012.922,155.029,-132.172,-27.427,38.959,-33.640
C06046=1012.927,154.789,-132.152,-27.413,38.831,-33.681
C06047=1012.932,154.549,-132.130,-27.399,38.702,-33.721
C06048=1012.937,154.308,-132.110,-27.385,38.574,-33.764
C06049=1012.941,154.067,-132.088,-27.370,38.445,-33.806
C06050=1012.945,153.827,-132.067,-27.356,38.317,-33.847
C06051=1012.950,153.585,-132.046,-27.341,38.188,-33.889
C06052=1012.955,153.344,-132.025,-27.327,38.059,-33.932
C06053=1012.960,153.103,-132.003,-27.312,37.930,-33.975
C06054=1012.964,152.862,-131.982,-27.297,37.803,-34.017
C06055=1012.969,152.620,-131.961,-27.282,37.674,-34.060
C06056=1012.974,152.378,-131.940,-27.267,37.546,-34.103
C06057=1012.979,152.135,-131.919,-27.252,37.416,-34.148
C06058=1012.983,151.886,-131.897,-27.236,37.284,-34.193
C06059=1012.989,151.630,-131.875,-27.220,37.150,-34.239
C06060=1012.993,151.369,-131.851,-27.204,37.011,-34.287
C06061=1012.999,151.097,-131.827,-27.186,36.868,-34.337
C06062=1013.004,150.819,-131.803,-27.169,36.722,-34.388
C06063=1013.010,150.533,-131.778,-27.150,36.571,-34.440
C06064=1013.016,150.240,-131.752,-27.131,36.417,-34.494
C06065=1013.021,149.943,-131.726,-27.112,36.261,-34.549
C06066=1013.027,149.644,-131.699,-27.092,36.105,-34.604
C06067=1013.033,149.344,-131.673,-27.072,35.947,-34.660
C06068=1013.039,149.045,-131.647,-27.052,35.791,-34.717
C06069=1013.044,148.748,-131.621,-27.032,35.635,-34.773
C06070=1013.051,148.457,-131.595,-27.013,35.484,-34.828
C06071=1013.056,148.172,-131.570,-26.993,35.335,-34.883
C06072=1013.061,147.895,-131.545,-26.974,35.189,-34.936
C06073=1013.067,147.624,-131.521,-26.956,35.049,-34.988
C06074=1013.072,147.363,-131.498,-26.937,34.913,-35.040
C06075=1013.077,147.109,-131.476,-26.920,34.781,-35.089
C06076=1013.082,146.861,-131.454,-26.902,34.652,-35.138
C06077=1013.086,146.617,-131.433,-26.885,34.527,-35.186
C06078=1013.092,146.375,-131.411,-26.868,34.402,-35.233
C06079=1013.097,146.133,-131.390,-26.851,34.276,-35.281
C06080=1013.101,145.890,-131.368,-26.834,34.152,-35.329
C06081=1013.106,145.649,-131.347,-26.816,34.027,-35.377
C06082=1013.111,145.407,-131.325,-26.799,33.903,-35.426
C06083=1013.116,145.165,-131.304,-26.781,33.778,-35.475
C06084=1013.120,144.924,-131.282,-26.764,33.656,-35.523
C06085=1013.125,144.682,-131.261,-26.746,33.532,-35.571
C06086=1013.131,144.370,-131.234,-26.723,33.372,-35.635
C06087=1013.140,143.958,-131.197,-26.693,33.163,-35.718
C06088=1013.144,143.718,-131.176,-26.675,33.041,-35.766
C06089=1013.149,143.477,-131.154,-26.657,32.919,-35.817
C06090=1013.154,143.237,-131.133,-26.639,32.797,-35.866
C06091=1013.158,142.997,-131.112,-26.621,32.676,-35.915
C06092=1013.163,142.757,-131.091,-26.603,32.554,-35.964
C06093=1013.168,142.518,-131.069,-26.584,32.434,-36.015
C06094=1013.173,142.277,-131.048,-26.566,32.313,-36.063
C06095=1013.178,142.038,-131.026,-26.548,32.193,-36.113
C06096=1013.182,141.800,-131.005,-26.529,32.073,-36.164
C06097=1013.187,141.561,-130.983,-26.511,31.953,-36.213
C06098=1013.192,141.316,-130.962,-26.492,31.831,-36.266
C06099=1013.196,141.105,-130.943,-26.475,31.725,-36.310
C06100=1013.201,140.849,-130.921,-26.455,31.598,-36.363
C06101=1013.204,140.677,-130.906,-26.442,31.513,-36.399
C06102=1013.212,140.305,-130.872,-26.412,31.327,-36.479
C06103=1013.217,140.030,-130.848,-26.390,31.190,-36.537
C06104=1013.224,139.735,-130.821,-26.366,31.044,-36.601
C06105=1013.229,139.427,-130.793,-26.342,30.892,-36.667
C06106=1013.236,139.114,-130.766,-26.316,30.738,-36.733
C06107=1013.242,138.807,-130.739,-26.291,30.586,-36.801
C06108=1013.247,138.513,-130.712,-26.267,30.442,-36.864
C06109=1013.253,138.239,-130.688,-26.244,30.308,-36.925
C06110=1013.258,137.987,-130.665,-26.224,30.185,-36.979
C06111=1013.266,137.567,-130.628,-26.189,29.980,-37.071
C06112=1013.274,137.183,-130.594,-26.156,29.792,-37.156
C06113=1013.282,136.767,-130.556,-26.121,29.591,-37.248
C06114=1013.290,136.384,-130.522,-26.088,29.404,-37.334
C06115=1013.298,135.998,-130.488,-26.055,29.219,-37.419
C06116=1013.306,135.579,-130.450,-26.019,29.017,-37.513
C06117=1013.311,135.355,-130.430,-26.000,28.910,-37.564
C06118=1013.315,135.122,-130.409,-25.979,28.797,-37.617
C06119=1013.321,134.837,-130.383,-25.955,28.662,-37.681
C06120=1013.326,134.540,-130.357,-25.929,28.520,-37.748
C06121=1013.331,134.302,-130.336,-25.907,28.406,-37.802
C06122=1013.336,134.067,-130.315,-25.886,28.294,-37.856
C06123=1013.340,133.832,-130.293,-25.865,28.183,-37.910
C06124=1013.344,133.597,-130.272,-25.845,28.072,-37.963
C06125=1013.350,133.361,-130.251,-25.823,27.960,-38.018
C06126=1013.355,133.127,-130.230,-25.802,27.849,-38.072
C06127=1013.359,132.891,-130.209,-25.781,27.738,-38.126
C06128=1013.363,132.656,-130.188,-25.759,27.627,-38.181
C06129=1013.368,132.422,-130.167,-25.738,27.518,-38.235
C06130=1013.375,132.065,-130.135,-25.706,27.351,-38.317
C06131=1013.382,131.716,-130.103,-25.673,27.187,-38.400
C06132=1013.387,131.481,-130.083,-25.652,27.077,-38.454
C06133=1013.391,131.246,-130.061,-25.630,26.968,-38.510
C06134=1013.396,131.011,-130.040,-25.608,26.859,-38.565
C06135=1013.401,130.776,-130.019,-25.586,26.750,-38.620
C06136=1013.405,130.541,-129.998,-25.563,26.641,-38.676
C06137=1013.409,130.306,-129.976,-25.541,26.532,-38.731
C06138=1013.414,130.071,-129.955,-25.519,26.424,-38.787
C06139=1013.419,129.836,-129.934,-25.497,26.316,-38.843
C06140=1013.424,129.601,-129.913,-25.474,26.207,-38.899
C06141=1013.428,129.366,-129.891,-25.452,26.099,-38.955
C06142=1013.432,129.131,-129.871,-25.429,25.992,-39.012
C06143=1013.437,128.896,-129.850,-25.406,25.885,-39.068
C06144=1013.442,128.661,-129.827,-25.384,25.777,-39.124
C06145=1013.446,128.426,-129.807,-25.361,25.671,-39.181
C06146=1013.451,128.191,-129.786,-25.338,25.563,-39.237
C06147=1013.456,127.957,-129.764,-25.315,25.457,-39.295
C06148=1013.460,127.721,-129.743,-25.292,25.351,-39.352
C06149=1013.465,127.486,-129.722,-25.269,25.245,-39.409
C06150=1013.469,127.251,-129.700,-25.245,25.138,-39.466
C06151=1013.474,127.016,-129.679,-25.222,25.032,-39.524
C06152=1013.478,126.781,-129.659,-25.199,24.927,-39.582
C06153=1013.483,126.547,-129.637,-25.175,24.822,-39.638
C06154=1013.488,126.311,-129.616,-25.152,24.717,-39.696
C06155=1013.492,126.076,-129.595,-25.128,24.612,-39.754
C06156=1013.497,125.841,-129.573,-25.104,24.506,-39.812
C06157=1013.501,125.606,-129.552,-25.080,24.402,-39.869
C06158=1013.505,125.371,-129.531,-25.056,24.298,-39.928
C06159=1013.511,125.136,-129.509,-25.032,24.194,-39.986
C06160=1013.515,124.901,-129.488,-25.008,24.090,-40.045
C06161=1013.520,124.667,-129.467,-24.984,23.986,-40.104
C06162=1013.524,124.431,-129.446,-24.960,23.883,-40.162
C06163=1013.528,124.196,-129.425,-24.936,23.780,-40.220
C06164=1013.534,123.962,-129.403,-24.911,23.676,-40.279
C06165=1013.538,123.726,-129.382,-24.887,23.574,-40.338
C06166=1013.542,123.492,-129.360,-24.862,23.470,-40.398
C06167=1013.547,123.257,-129.340,-24.837,23.368,-40.457
C06168=1013.551,123.022,-129.318,-24.813,23.266,-40.515
C06169=1013.555,122.787,-129.297,-24.788,23.164,-40.574
C06170=1013.560,122.552,-129.275,-24.763,23.063,-40.635
C06171=1013.565,122.317,-129.254,-24.738,22.961,-40.695
C06172=1013.569,122.082,-129.233,-24.713,22.860,-40.754
C06173=1013.574,121.848,-129.212,-24.688,22.759,-40.814
C06174=1013.578,121.612,-129.190,-24.663,22.658,-40.874
C06175=1013.583,121.377,-129.168,-24.638,22.557,-40.933
C06176=1013.588,121.143,-129.148,-24.612,22.457,-40.994
C06177=1013.591,120.907,-129.126,-24.587,22.356,-41.054
C06178=1013.596,120.673,-129.105,-24.561,22.257,-41.115
C06179=1013.600,120.438,-129.083,-24.534,22.150,-41.179
C06180=1013.606,120.203,-129.062,-24.506,22.042,-41.244
C06181=1013.611,119.968,-129.041,-24.478,21.932,-41.311
C06182=1013.635,118.771,-128.933,-24.343,21.420,-41.628
C06183=1013.639,118.576,-128.916,-24.343,21.420,-41.629
C06184=1013.647,118.178,-128.880,-24.342,21.420,-41.633
C06185=1013.655,117.779,-128.844,-24.342,21.420,-41.637
C06186=1013.663,117.381,-128.808,-24.341,21.420,-41.638
C06187=1013.670,116.983,-128.772,-24.341,21.421,-41.642
C06188=1013.678,116.584,-128.736,-24.340,21.420,-41.646
C06189=1013.686,116.185,-128.701,-24.340,21.421,-41.649
C06190=1013.694,115.788,-128.664,-24.340,21.422,-41.652
C06191=1013.702,115.390,-128.629,-24.339,21.422,-41.655
C06192=1013.710,114.990,-128.593,-24.339,21.422,-41.659
C06193=1013.718,114.592,-128.556,-24.338,21.422,-41.662
C06194=1013.726,114.194,-128.520,-24.338,21.423,-41.664
C06195=1013.733,113.796,-128.484,-24.337,21.422,-41.668
C06196=1013.740,113.398,-128.449,-24.337,21.423,-41.671
C06197=1013.748,113.000,-128.412,-24.336,21.423,-41.675
C06198=1013.756,112.601,-128.377,-24.336,21.423,-41.677
C06199=1013.764,112.203,-128.340,-24.335,21.424,-41.681
C06200=1013.770,111.804,-128.305,-24.335,21.423,-41.684
C06201=1013.778,111.406,-128.269,-24.334,21.424,-41.688
C06202=1013.786,111.008,-128.233,-24.334,21.425,-41.690
C06203=1013.792,110.609,-128.196,-24.334,21.425,-41.694
C06204=1013.800,110.211,-128.161,-24.333,21.425,-41.697
C06205=1013.808,109.813,-128.124,-24.333,21.425,-41.701
C06206=1013.815,109.414,-128.089,-24.332,21.426,-41.703
C06207=1013.822,109.016,-128.052,-24.332,21.426,-41.707
C06208=1013.829,108.617,-128.017,-24.331,21.426,-41.710
C06209=1013.837,108.219,-127.980,-24.331,21.426,-41.714
C06210=1013.843,107.820,-127.945,-24.330,21.426,-41.717
C06211=1013.851,107.422,-127.909,-24.330,21.427,-41.719
C06212=1013.857,107.024,-127.872,-24.330,21.427,-41.723
C06213=1013.865,106.625,-127.837,-24.329,21.427,-41.727
C06214=1013.872,106.227,-127.800,-24.328,21.427,-41.730
C06215=1013.879,105.827,-127.764,-24.328,21.428,-41.734
C06216=1013.886,105.430,-127.728,-24.328,21.428,-41.736
C06217=1013.892,105.032,-127.692,-24.327,21.429,-41.740
C06218=1013.900,104.632,-127.656,-24.327,21.429,-41.743
C06219=1013.907,104.235,-127.620,-24.326,21.429,-41.747
C06220=1013.913,103.836,-127.585,-24.326,21.429,-41.751
C06221=1013.921,103.437,-127.548,-24.325,21.430,-41.754
C06222=1013.927,103.039,-127.512,-24.325,21.430,-41.756
C06223=1013.934,102.640,-127.476,-24.324,21.430,-41.760
C06224=1013.940,102.241,-127.440,-24.324,21.430,-41.763
C06225=1013.946,101.843,-127.404,-24.323,21.430,-41.767
C06226=1013.954,101.444,-127.368,-24.323,21.431,-41.771
C06227=1013.960,101.045,-127.332,-24.322,21.431,-41.775
C06228=1013.966,100.647,-127.295,-24.322,21.431,-41.778
C06229=1013.973,100.248,-127.260,-24.322,21.432,-41.780
C06230=1013.979,99.850,-127.224,-24.321,21.432,-41.784
C06231=1013.986,99.451,-127.187,-24.320,21.432,-41.787
C06232=1013.992,99.052,-127.152,-24.320,21.432,-41.791
C06233=1013.999,98.654,-127.116,-24.319,21.433,-41.795
C06234=1014.006,98.255,-127.079,-24.319,21.432,-41.798
C06235=1014.012,97.856,-127.043,-24.318,21.433,-41.802
C06236=1014.018,97.457,-127.007,-24.318,21.433,-41.806
C06237=1014.024,97.059,-126.971,-24.318,21.434,-41.808
C06238=1014.031,96.660,-126.935,-24.317,21.434,-41.811
C06239=1014.037,96.261,-126.899,-24.317,21.435,-41.815
C06240=1014.042,95.863,-126.863,-24.316,21.435,-41.819
C06241=1014.049,95.464,-126.827,-24.316,21.435,-41.822
C06242=1014.055,95.065,-126.791,-24.315,21.435,-41.826
C06243=1014.061,94.667,-126.755,-24.315,21.436,-41.830
C06244=1014.067,94.267,-126.719,-24.314,21.435,-41.833
C06245=1014.074,93.869,-126.683,-24.313,21.436,-41.837
C06246=1014.079,93.469,-126.646,-24.313,21.436,-41.841
C06247=1014.086,93.071,-126.611,-24.312,21.437,-41.844
C06248=1014.091,92.672,-126.575,-24.312,21.437,-41.846
C06249=1014.097,92.273,-126.538,-24.312,21.437,-41.850
C06250=1014.103,91.874,-126.503,-24.311,21.438,-41.854
C06251=1014.109,91.475,-126.466,-24.311,21.438,-41.857
C06252=1014.115,91.076,-126.429,-24.310,21.438,-41.861
C06253=1014.121,90.677,-126.394,-24.310,21.438,-41.865
C06254=1014.126,90.278,-126.358,-24.309,21.439,-41.868
C06255=1014.132,89.878,-126.322,-24.309,21.439,-41.872
C06256=1014.138,89.481,-126.286,-24.308,21.439,-41.875
C06257=1014.143,89.088,-126.251,-24.308,21.439,-41.879
C06258=1014.149,88.701,-126.215,-24.307,21.440,-41.883
C06259=1014.154,88.319,-126.180,-24.307,21.440,-41.887
C06260=1014.160,87.935,-126.146,-24.306,21.440,-41.890
C06261=1014.165,87.547,-126.111,-24.305,21.440,-41.894
C06262=1014.171,87.151,-126.076,-24.305,21.441,-41.898
C06263=1014.176,86.748,-126.039,-24.304,21.441,-41.901
C06264=1014.182,86.343,-126.002,-24.304,21.442,-41.905
C06265=1014.188,85.935,-125.965,-24.303,21.441,-41.908
C06266=1014.193,85.527,-125.929,-24.303,21.442,-41.912
C06267=1014.199,85.115,-125.891,-24.302,21.442,-41.916
C06268=1014.204,84.703,-125.855,-24.302,21.443,-41.920
C06269=1014.209,84.290,-125.817,-24.301,21.443,-41.923
C06270=1014.215,83.874,-125.779,-24.301,21.443,-41.927
C06271=1014.221,83.457,-125.742,-24.300,21.444,-41.931
C06272=1014.227,83.038,-125.704,-24.300,21.444,-41.935
C06273=1014.232,82.618,-125.666,-24.299,21.444,-41.938
C06274=1014.238,82.196,-125.628,-24.299,21.444,-41.942
C06275=1014.240,81.985,-125.609,-24.299,21.445,-41.944
C06276=1014.243,81.774,-125.590,-24.298,21.444,-41.947
C06277=1014.246,81.562,-125.571,-24.298,21.445,-41.949
C06278=1014.249,81.350,-125.552,-24.298,21.445,-41.951
C06279=1014.251,81.138,-125.533,-24.297,21.445,-41.953
C06280=1014.254,80.925,-125.513,-24.297,21.445,-41.955
C06281=1014.257,80.713,-125.494,-24.297,21.445,-41.956
C06282=1014.260,80.500,-125.475,-24.297,21.446,-41.958
C06283=1014.262,80.287,-125.457,-24.296,21.446,-41.960
C06284=1014.265,80.075,-125.437,-24.296,21.446,-41.962
C06285=1014.268,79.863,-125.418,-24.296,21.446,-41.964
C06286=1014.270,79.653,-125.398,-24.296,21.447,-41.966
C06287=1014.276,79.239,-125.361,-24.295,21.447,-41.970
C06288=1014.281,78.833,-125.325,-24.294,21.447,-41.973
C06289=1014.285,78.436,-125.289,-24.294,21.447,-41.977
C06290=1014.290,78.046,-125.254,-24.293,21.448,-41.980
C06291=1014.295,77.659,-125.219,-24.293,21.447,-41.986
C06292=1014.301,77.273,-125.184,-24.292,21.448,-41.989
C06293=1014.304,76.885,-125.149,-24.292,21.449,-41.994
C06294=1014.310,76.490,-125.114,-24.291,21.449,-41.997
C06295=1014.315,76.088,-125.078,-24.291,21.449,-42.001
C06296=1014.319,75.677,-125.041,-24.290,21.450,-42.004
C06297=1014.324,75.257,-125.003,-24.290,21.450,-42.008
C06298=1014.327,75.045,-124.984,-24.289,21.451,-42.010
C06299=1014.329,74.831,-124.964,-24.289,21.451,-42.012
C06300=1014.332,74.618,-124.945,-24.289,21.450,-42.015
C06301=1014.335,74.404,-124.925,-24.288,21.451,-42.017
C06302=1014.337,74.191,-124.907,-24.288,21.451,-42.019
C06303=1014.339,73.978,-124.888,-24.288,21.451,-42.021
C06304=1014.342,73.766,-124.869,-24.288,21.451,-42.023
C06305=1014.344,73.555,-124.850,-24.287,21.452,-42.025
C06306=1014.349,73.135,-124.812,-24.287,21.452,-42.028
C06307=1014.354,72.717,-124.774,-24.286,21.452,-42.034
C06308=1014.359,72.301,-124.737,-24.285,21.452,-42.037
C06309=1014.363,71.888,-124.700,-24.285,21.453,-42.041
C06310=1014.369,71.476,-124.663,-24.285,21.453,-42.045
C06311=1014.373,71.065,-124.626,-24.284,21.454,-42.049
C06312=1014.378,70.655,-124.589,-24.283,21.453,-42.054
C06313=1014.383,70.244,-124.552,-24.283,21.454,-42.058
C06314=1014.387,69.832,-124.515,-24.282,21.454,-42.061
C06315=1014.391,69.422,-124.478,-24.282,21.455,-42.065
C06316=1014.396,69.011,-124.442,-24.281,21.455,-42.069
C06317=1014.400,68.602,-124.405,-24.280,21.455,-42.074
C06318=1014.405,68.195,-124.368,-24.280,21.456,-42.078
C06319=1014.409,67.789,-124.332,-24.279,21.456,-42.082
C06320=1014.414,67.385,-124.296,-24.279,21.457,-42.085
C06321=1014.418,66.981,-124.260,-24.278,21.457,-42.089
C06322=1014.422,66.579,-124.224,-24.278,21.457,-42.094
C06323=1014.427,66.178,-124.188,-24.277,21.457,-42.098
C06324=1014.430,65.780,-124.152,-24.277,21.458,-42.102
C06325=1014.435,65.373,-124.115,-24.276,21.458,-42.106
C06326=1014.437,65.160,-124.096,-24.276,21.459,-42.108
C06327=1014.439,64.939,-124.077,-24.275,21.458,-42.111
C06328=1014.442,64.708,-124.056,-24.275,21.458,-42.113
C06329=1014.445,64.473,-124.035,-24.275,21.459,-42.115
C06330=1014.446,64.236,-124.014,-24.274,21.459,-42.116
C06331=1014.449,64.007,-123.993,-24.274,21.459,-42.120
C06332=1014.451,63.789,-123.973,-24.274,21.460,-42.122
C06333=1014.453,63.582,-123.955,-24.274,21.460,-42.124
C06334=1014.455,63.365,-123.936,-24.273,21.459,-42.127
C06335=1014.458,63.116,-123.914,-24.273,21.460,-42.129
C06336=1014.461,62.848,-123.890,-24.272,21.460,-42.131
C06337=1014.463,62.595,-123.867,-24.272,21.460,-42.133
C06338=1014.467,62.175,-123.830,-24.271,21.461,-42.139
C06339=1014.472,61.775,-123.794,-24.271,21.461,-42.142
C06340=1014.475,61.375,-123.758,-24.270,21.462,-42.146
C06341=1014.479,60.975,-123.722,-24.270,21.462,-42.150
C06342=1014.483,60.575,-123.687,-24.269,21.462,-42.155
C06343=1014.487,60.174,-123.651,-24.269,21.463,-42.159
C06344=1014.491,59.775,-123.615,-24.268,21.463,-42.163
C06345=1014.495,59.374,-123.579,-24.268,21.464,-42.166
C06346=1014.499,58.974,-123.544,-24.267,21.463,-42.172
C06347=1014.502,58.574,-123.508,-24.266,21.464,-42.175
C06348=1014.506,58.174,-123.472,-24.266,21.464,-42.179
C06349=1014.510,57.774,-123.437,-24.265,21.465,-42.183
C06350=1014.513,57.374,-123.401,-24.264,21.465,-42.188
C06351=1014.517,56.973,-123.365,-24.264,21.465,-42.192
C06352=1014.521,56.574,-123.330,-24.264,21.466,-42.196
C06353=1014.525,56.173,-123.294,-24.263,21.465,-42.201
C06354=1014.528,55.773,-123.258,-24.262,21.467,-42.205
C06355=1014.532,55.373,-123.223,-24.262,21.467,-42.209
C06356=1014.536,54.973,-123.187,-24.261,21.468,-42.212
C06357=1014.539,54.573,-123.151,-24.260,21.468,-42.218
C06358=1014.543,54.173,-123.116,-24.260,21.468,-42.221
C06359=1014.546,53.773,-123.081,-24.259,21.468,-42.225
C06360=1014.549,53.373,-123.044,-24.259,21.468,-42.230
C06361=1014.553,52.972,-123.009,-24.258,21.469,-42.234
C06362=1014.557,52.572,-122.974,-24.258,21.469,-42.238
C06363=1014.560,52.172,-122.939,-24.257,21.469,-42.243
C06364=1014.563,51.772,-122.902,-24.256,21.470,-42.247
C06365=1014.566,51.372,-122.867,-24.256,21.471,-42.251
C06366=1014.570,50.971,-122.832,-24.255,21.471,-42.255
C06367=1014.573,50.572,-122.796,-24.255,21.471,-42.260
C06368=1014.577,50.172,-122.761,-24.254,21.472,-42.264
C06369=1014.580,49.771,-122.725,-24.254,21.472,-42.268
C06370=1014.583,49.371,-122.689,-24.253,21.472,-42.273
C06371=1014.586,48.971,-122.654,-24.252,21.473,-42.277
C06372=1014.590,48.571,-122.619,-24.251,21.472,-42.282
C06373=1014.593,48.172,-122.583,-24.251,21.474,-42.286
C06374=1014.596,47.771,-122.548,-24.251,21.474,-42.290
C06375=1014.599,47.371,-122.513,-24.250,21.474,-42.295
C06376=1014.602,46.971,-122.477,-24.249,21.475,-42.299
C06377=1014.605,46.571,-122.441,-24.249,21.475,-42.302
C06378=1014.609,46.171,-122.407,-24.248,21.475,-42.308
C06379=1014.612,45.771,-122.371,-24.247,21.475,-42.311
C06380=1014.615,45.371,-122.335,-24.247,21.477,-42.316
C06381=1014.618,44.971,-122.300,-24.246,21.477,-42.321
C06382=1014.621,44.571,-122.264,-24.246,21.477,-42.325
C06383=1014.623,44.171,-122.230,-24.245,21.477,-42.330
C06384=1014.627,43.770,-122.194,-24.244,21.477,-42.333
C06385=1014.630,43.371,-122.159,-24.244,21.479,-42.338
C06386=1014.632,42.971,-122.124,-24.243,21.479,-42.343
C06387=1014.636,42.571,-122.089,-24.243,21.479,-42.347
C06388=1014.638,42.171,-122.053,-24.242,21.479,-42.352
C06389=1014.641,41.771,-122.018,-24.241,21.479,-42.356
C06390=1014.644,41.371,-121.982,-24.241,21.480,-42.359
C06391=1014.646,40.971,-121.948,-24.240,21.481,-42.365
C06392=1014.649,40.571,-121.913,-24.240,21.481,-42.369
C06393=1014.652,40.171,-121.877,-24.239,21.481,-42.374
C06394=1014.655,39.772,-121.842,-24.238,21.481,-42.378
C06395=1014.658,39.372,-121.807,-24.238,21.482,-42.383
C06396=1014.660,38.972,-121.772,-24.237,21.483,-42.387
C06397=1014.663,38.572,-121.737,-24.237,21.483,-42.391
C06398=1014.665,38.172,-121.701,-24.236,21.483,-42.396
C06399=1014.669,37.772,-121.666,-24.235,21.483,-42.400
C06400=1014.671,37.372,-121.631,-24.235,21.484,-42.405
C06401=1014.674,36.972,-121.596,-24.234,21.485,-42.409
C06402=1014.677,36.573,-121.561,-24.233,21.484,-42.414
C06403=1014.679,36.173,-121.526,-24.233,21.485,-42.418
C06404=1014.682,35.773,-121.491,-24.232,21.486,-42.424
C06405=1014.683,35.374,-121.456,-24.231,21.486,-42.428
C06406=1014.686,34.973,-121.421,-24.231,21.486,-42.433
C06407=1014.688,34.574,-121.386,-24.230,21.486,-42.437
C06408=1014.691,34.174,-121.351,-24.229,21.487,-42.442
C06409=1014.694,33.775,-121.316,-24.229,21.488,-42.446
C06410=1014.696,33.375,-121.281,-24.228,21.487,-42.451
C06411=1014.698,32.976,-121.246,-24.228,21.489,-42.455
C06412=1014.701,32.575,-121.211,-24.227,21.489,-42.461
C06413=1014.703,32.176,-121.176,-24.226,21.489,-42.464
C06414=1014.705,31.776,-121.141,-24.226,21.489,-42.469
C06415=1014.707,31.377,-121.106,-24.225,21.490,-42.474
C06416=1014.710,30.977,-121.072,-24.224,21.490,-42.479
C06417=1014.712,30.578,-121.037,-24.224,21.491,-42.483
C06418=1014.715,30.178,-121.002,-24.223,21.491,-42.488
C06419=1014.716,29.778,-120.967,-24.223,21.492,-42.492
C06420=1014.719,29.378,-120.932,-24.222,21.492,-42.497
C06421=1014.721,28.980,-120.897,-24.221,21.492,-42.501
C06422=1014.723,28.581,-120.862,-24.221,21.493,-42.507
C06423=1014.725,28.180,-120.828,-24.220,21.493,-42.510
C06424=1014.727,27.781,-120.793,-24.219,21.493,-42.516
C06425=1014.729,27.381,-120.759,-24.219,21.495,-42.520
C06426=1014.732,26.983,-120.723,-24.218,21.494,-42.525
C06427=1014.733,26.583,-120.688,-24.218,21.495,-42.529
C06428=1014.735,26.184,-120.654,-24.217,21.496,-42.534
C06429=1014.737,25.784,-120.619,-24.216,21.496,-42.540
C06430=1014.739,25.385,-120.585,-24.215,21.496,-42.543
C06431=1014.742,24.986,-120.550,-24.215,21.497,-42.549
C06432=1014.743,24.586,-120.515,-24.214,21.497,-42.553
C06433=1014.746,24.187,-120.481,-24.213,21.497,-42.558
C06434=1014.747,23.804,-120.448,-24.213,21.498,-42.562
C06435=1014.748,23.474,-120.419,-24.213,21.498,-42.564
C06436=1014.750,23.202,-120.395,-24.212,21.498,-42.567
C06437=1014.751,22.968,-120.375,-24.211,21.499,-42.573
C06438=1014.752,22.735,-120.355,-24.211,21.500,-42.577
C06439=1014.752,22.470,-120.332,-24.211,21.500,-42.580
C06440=1014.755,22.148,-120.304,-24.210,21.500,-42.584
C06441=1014.756,21.773,-120.271,-24.210,21.501,-42.586
C06442=1014.758,21.359,-120.236,-24.209,21.501,-42.593
C06443=1014.759,21.116,-120.215,-24.208,21.501,-42.597
C06444=1014.760,20.843,-120.192,-24.208,21.502,-42.599
C06445=1014.761,20.551,-120.166,-24.207,21.501,-42.602
C06446=1014.763,20.255,-120.140,-24.207,21.501,-42.604
C06447=1014.763,19.967,-120.116,-24.207,21.503,-42.606
C06448=1014.766,19.702,-120.093,-24.206,21.502,-42.610
C06449=1014.766,19.465,-120.072,-24.206,21.503,-42.613
C06450=1014.767,19.255,-120.054,-24.205,21.503,-42.617
C06451=1014.769,18.857,-120.020,-24.205,21.503,-42.622
C06452=1014.770,18.460,-119.986,-24.204,21.503,-42.626
C06453=1014.772,18.065,-119.952,-24.203,21.504,-42.632
C06454=1014.773,17.670,-119.918,-24.203,21.505,-42.635
C06455=1014.774,17.276,-119.883,-24.202,21.505,-42.641
C06456=1014.777,16.882,-119.850,-24.201,21.505,-42.646
C06457=1014.778,16.490,-119.816,-24.201,21.506,-42.650
C06458=1014.779,16.098,-119.782,-24.200,21.506,-42.656
C06459=1014.781,15.707,-119.749,-24.200,21.507,-42.659
C06460=1014.782,15.317,-119.715,-24.199,21.507,-42.665
C06461=1014.783,14.928,-119.682,-24.198,21.508,-42.670
C06462=1014.785,14.538,-119.648,-24.198,21.508,-42.674
C06463=1014.786,14.150,-119.615,-24.197,21.509,-42.680
C06464=1014.787,13.762,-119.582,-24.196,21.509,-42.683
C06465=1014.788,13.375,-119.549,-24.196,21.509,-42.689
C06466=1014.790,12.989,-119.516,-24.195,21.511,-42.693
C06467=1014.791,12.602,-119.482,-24.194,21.510,-42.698
C06468=1014.793,12.216,-119.449,-24.193,21.510,-42.703
C06469=1014.794,11.829,-119.416,-24.193,21.512,-42.707
C06470=1014.795,11.442,-119.383,-24.192,21.511,-42.713
C06471=1014.796,11.057,-119.350,-24.192,21.512,-42.716
C06472=1014.797,10.674,-119.318,-24.191,21.513,-42.722
C06473=1014.799,10.293,-119.285,-24.191,21.513,-42.726
C06474=1014.799,9.915,-119.252,-24.190,21.513,-42.731
C06475=1014.801,9.538,-119.220,-24.189,21.514,-42.737
C06476=1014.802,9.163,-119.189,-24.189,21.514,-42.740
C06477=1014.803,8.786,-119.157,-24.188,21.515,-42.746
C06478=1014.803,8.408,-119.124,-24.187,21.515,-42.751
C06479=1014.805,8.027,-119.091,-24.187,21.516,-42.755
C06480=1014.806,7.643,-119.059,-24.186,21.516,-42.761
C06481=1014.807,7.256,-119.026,-24.185,21.517,-42.764
C06482=1014.808,6.865,-118.992,-24.185,21.517,-42.770
C06483=1014.808,6.473,-118.959,-24.184,21.517,-42.775
C06484=1014.810,6.080,-118.926,-24.183,21.519,-42.779
C06485=1014.811,5.686,-118.892,-24.182,21.518,-42.785
C06486=1014.812,5.292,-118.859,-24.182,21.519,-42.790
C06487=1014.812,4.897,-118.825,-24.181,21.520,-42.794
C06488=1014.813,4.501,-118.791,-24.180,21.519,-42.799
C06489=1014.814,4.106,-118.758,-24.180,21.520,-42.805
C06490=1014.814,3.716,-118.725,-24.179,21.521,-42.809
C06491=1014.816,3.357,-118.694,-24.179,21.521,-42.812
C06492=1014.816,3.029,-118.667,-24.178,21.521,-42.817
C06493=1014.817,2.716,-118.640,-24.177,21.522,-42.823
C06494=1014.818,2.393,-118.613,-24.177,21.522,-42.827
C06495=1014.818,2.040,-118.582,-24.176,21.523,-42.833
C06496=1014.819,1.655,-118.550,-24.175,21.524,-42.836
C06497=1014.820,1.256,-118.516,-24.175,21.523,-42.841
C06498=1014.820,0.858,-118.483,-24.174,21.525,-42.846
C06499=1014.821,0.458,-118.449,-24.173,21.525,-42.851
C06500=1014.821,0.056,-118.415,-24.173,21.525,-42.857
C06501=1014.822,-0.347,-118.381,-24.172,21.525,-42.862
C06502=1014.823,-0.754,-118.347,-24.171,21.526,-42.867
C06503=1014.824,-1.161,-118.313,-24.171,21.527,-42.872
C06504=1014.824,-1.572,-118.278,-24.170,21.527,-42.877
C06505=1014.824,-1.984,-118.243,-24.169,21.528,-42.882
C06506=1014.825,-2.399,-118.208,-24.169,21.529,-42.888
C06507=1014.825,-2.816,-118.173,-24.168,21.529,-42.893
C06508=1014.826,-3.235,-118.137,-24.167,21.529,-42.899
C06509=1014.826,-3.656,-118.102,-24.166,21.530,-42.904
C06510=1014.827,-3.868,-118.084,-24.166,21.530,-42.908
C06511=1014.827,-4.080,-118.066,-24.165,21.530,-42.910
C06512=1014.827,-4.294,-118.048,-24.165,21.530,-42.913
C06513=1014.828,-4.509,-118.030,-24.165,21.531,-42.915
C06514=1014.827,-4.725,-118.012,-24.164,21.531,-42.919
C06515=1014.828,-4.944,-117.994,-24.164,21.531,-42.921
C06516=1014.828,-5.164,-117.975,-24.163,21.532,-42.925
C06517=1014.828,-5.386,-117.957,-24.163,21.532,-42.927
C06518=1014.828,-5.608,-117.938,-24.163,21.532,-42.930
C06519=1014.828,-5.832,-117.919,-24.162,21.532,-42.934
C06520=1014.828,-6.055,-117.901,-24.162,21.533,-42.935
C06521=1014.829,-6.280,-117.882,-24.161,21.533,-42.939
C06522=1014.829,-6.505,-117.863,-24.161,21.533,-42.941
C06523=1014.829,-6.728,-117.844,-24.161,21.533,-42.944
C06524=1014.829,-6.952,-117.826,-24.160,21.534,-42.947
C06525=1014.829,-7.174,-117.807,-24.160,21.534,-42.950
C06526=1014.830,-7.395,-117.788,-24.160,21.535,-42.952
C06527=1014.829,-7.616,-117.770,-24.159,21.534,-42.956
C06528=1014.830,-7.835,-117.752,-24.159,21.535,-42.959
C06529=1014.830,-8.053,-117.733,-24.158,21.535,-42.961
C06530=1014.830,-8.270,-117.715,-24.158,21.536,-42.965
C06531=1014.830,-8.487,-117.697,-24.158,21.536,-42.967
C06532=1014.830,-8.704,-117.679,-24.157,21.536,-42.971
C06533=1014.831,-8.921,-117.661,-24.157,21.537,-42.973
C06534=1014.830,-9.137,-117.643,-24.156,21.536,-42.976
C06535=1014.831,-9.353,-117.625,-24.156,21.537,-42.980
C06536=1014.830,-9.570,-117.607,-24.156,21.537,-42.982
C06537=1014.831,-9.786,-117.589,-24.155,21.538,-42.985
C06538=1014.830,-10.002,-117.570,-24.155,21.538,-42.987
C06539=1014.831,-10.218,-117.553,-24.154,21.538,-42.991
C06540=1014.831,-10.434,-117.534,-24.154,21.539,-42.993
C06541=1014.830,-10.649,-117.517,-24.154,21.538,-42.996
C06542=1014.831,-10.864,-117.499,-24.153,21.539,-42.998
C06543=1014.830,-11.078,-117.481,-24.153,21.539,-43.002
C06544=1014.831,-11.293,-117.463,-24.152,21.539,-43.006
C06545=1014.831,-11.507,-117.446,-24.152,21.540,-43.007
C06546=1014.831,-11.720,-117.427,-24.152,21.540,-43.011
C06547=1014.830,-11.933,-117.410,-24.151,21.540,-43.013
C06548=1014.830,-12.145,-117.392,-24.151,21.540,-43.016
C06549=1014.830,-12.357,-117.374,-24.151,21.541,-43.019
C06550=1014.831,-12.568,-117.356,-24.150,21.541,-43.022
C06551=1014.830,-12.779,-117.339,-24.150,21.542,-43.024
C06552=1014.831,-13.199,-117.304,-24.149,21.542,-43.029
C06553=1014.830,-13.617,-117.270,-24.148,21.543,-43.035
C06554=1014.830,-14.030,-117.236,-24.148,21.543,-43.041
C06555=1014.830,-14.442,-117.201,-24.147,21.544,-43.046
C06556=1014.830,-14.851,-117.168,-24.146,21.544,-43.052
C06557=1014.830,-15.256,-117.134,-24.145,21.545,-43.057
C06558=1014.829,-15.659,-117.100,-24.145,21.545,-43.063
C06559=1014.829,-16.060,-117.067,-24.144,21.546,-43.068
C06560=1014.829,-16.460,-117.034,-24.143,21.546,-43.074
C06561=1014.828,-16.858,-117.001,-24.142,21.547,-43.079
C06562=1014.828,-17.256,-116.968,-24.142,21.548,-43.085
C06563=1014.828,-17.654,-116.935,-24.141,21.547,-43.090
C06564=1014.827,-18.065,-116.901,-24.140,21.548,-43.098
C06565=1014.827,-18.313,-116.880,-24.139,21.549,-43.101
C06566=1014.827,-18.600,-116.857,-24.139,21.549,-43.105
C06567=1014.826,-18.912,-116.831,-24.139,21.550,-43.107
C06568=1014.827,-19.224,-116.806,-24.139,21.550,-43.109
C06569=1014.826,-19.511,-116.781,-24.138,21.550,-43.113
C06570=1014.826,-19.761,-116.761,-24.138,21.551,-43.116
C06571=1014.826,-20.171,-116.727,-24.136,21.551,-43.123
C06572=1014.825,-20.570,-116.694,-24.136,21.552,-43.129
C06573=1014.824,-20.967,-116.662,-24.135,21.553,-43.135
C06574=1014.824,-21.364,-116.629,-24.134,21.552,-43.140
C06575=1014.823,-21.762,-116.596,-24.134,21.553,-43.146
C06576=1014.823,-22.160,-116.564,-24.133,21.554,-43.151
C06577=1014.822,-22.557,-116.531,-24.132,21.554,-43.156
C06578=1014.822,-22.955,-116.499,-24.131,21.555,-43.162
C06579=1014.820,-23.352,-116.465,-24.131,21.555,-43.168
C06580=1014.820,-23.750,-116.433,-24.130,21.556,-43.173
C06581=1014.819,-24.147,-116.400,-24.129,21.556,-43.178
C06582=1014.818,-24.545,-116.368,-24.128,21.557,-43.184
C06583=1014.818,-24.942,-116.335,-24.128,21.558,-43.190
C06584=1014.817,-25.340,-116.303,-24.127,21.558,-43.195
C06585=1014.816,-25.737,-116.270,-24.126,21.558,-43.201
C06586=1014.815,-26.135,-116.238,-24.125,21.559,-43.206
C06587=1014.815,-26.532,-116.205,-24.125,21.560,-43.212
C06588=1014.813,-26.930,-116.172,-24.124,21.560,-43.217
C06589=1014.813,-27.327,-116.140,-24.123,21.561,-43.221
C06590=1014.812,-27.724,-116.108,-24.123,21.562,-43.227
C06591=1014.810,-28.122,-116.075,-24.122,21.562,-43.232
C06592=1014.810,-28.519,-116.043,-24.121,21.562,-43.238
C06593=1014.808,-28.917,-116.010,-24.120,21.563,-43.243
C06594=1014.808,-29.314,-115.978,-24.120,21.564,-43.249
C06595=1014.807,-29.712,-115.946,-24.119,21.565,-43.255
C06596=1014.805,-30.110,-115.913,-24.118,21.565,-43.260
C06597=1014.805,-30.507,-115.881,-24.117,21.565,-43.265
C06598=1014.803,-30.905,-115.849,-24.117,21.566,-43.271
C06599=1014.802,-31.301,-115.816,-24.116,21.567,-43.277
C06600=1014.801,-31.699,-115.784,-24.115,21.568,-43.282
C06601=1014.800,-32.097,-115.751,-24.114,21.567,-43.287
C06602=1014.799,-32.494,-115.720,-24.114,21.568,-43.293
C06603=1014.797,-32.892,-115.687,-24.113,21.569,-43.299
C06604=1014.796,-33.289,-115.655,-24.112,21.570,-43.304
C06605=1014.795,-33.687,-115.622,-24.111,21.570,-43.310
C06606=1014.794,-34.084,-115.591,-24.111,21.570,-43.315
C06607=1014.792,-34.482,-115.558,-24.110,21.571,-43.321
C06608=1014.791,-34.879,-115.526,-24.109,21.571,-43.328
C06609=1014.790,-35.276,-115.494,-24.108,21.572,-43.334
C06610=1014.789,-35.674,-115.462,-24.107,21.572,-43.339
C06611=1014.787,-36.071,-115.430,-24.107,21.573,-43.344
C06612=1014.786,-36.469,-115.398,-24.106,21.573,-43.350
C06613=1014.784,-36.866,-115.366,-24.105,21.574,-43.356
C06614=1014.782,-37.263,-115.333,-24.105,21.575,-43.361
C06615=1014.781,-37.660,-115.301,-24.104,21.575,-43.366
C06616=1014.779,-38.057,-115.269,-24.103,21.576,-43.372
C06617=1014.778,-38.455,-115.237,-24.102,21.576,-43.378
C06618=1014.776,-38.852,-115.205,-24.102,21.577,-43.383
C06619=1014.774,-39.250,-115.173,-24.101,21.578,-43.389
C06620=1014.772,-39.647,-115.142,-24.100,21.578,-43.394
C06621=1014.771,-40.045,-115.109,-24.099,21.579,-43.400
C06622=1014.769,-40.442,-115.077,-24.099,21.579,-43.405
C06623=1014.767,-40.839,-115.045,-24.098,21.580,-43.411
C06624=1014.766,-41.236,-115.014,-24.097,21.581,-43.417
C06625=1014.764,-41.634,-114.982,-24.096,21.582,-43.422
C06626=1014.762,-42.031,-114.950,-24.096,21.582,-43.427
C06627=1014.760,-42.429,-114.918,-24.095,21.582,-43.433
C06628=1014.758,-42.825,-114.886,-24.094,21.583,-43.439
C06629=1014.756,-43.222,-114.854,-24.093,21.584,-43.444
C06630=1014.754,-43.620,-114.822,-24.092,21.584,-43.451
C06631=1014.753,-44.017,-114.791,-24.092,21.585,-43.457
C06632=1014.750,-44.415,-114.759,-24.091,21.585,-43.462
C06633=1014.749,-44.812,-114.727,-24.090,21.585,-43.468
C06634=1014.747,-45.209,-114.695,-24.089,21.586,-43.473
C06635=1014.744,-45.607,-114.664,-24.089,21.587,-43.479
C06636=1014.742,-46.003,-114.632,-24.088,21.588,-43.485
C06637=1014.740,-46.401,-114.600,-24.087,21.589,-43.490
C06638=1014.738,-46.798,-114.569,-24.086,21.588,-43.496
C06639=1014.736,-47.195,-114.537,-24.086,21.589,-43.501
C06640=1014.734,-47.592,-114.505,-24.085,21.590,-43.507
C06641=1014.731,-47.989,-114.474,-24.084,21.591,-43.512
C06642=1014.729,-48.387,-114.442,-24.084,21.592,-43.518
C06643=1014.726,-48.784,-114.410,-24.083,21.592,-43.525
C06644=1014.725,-49.181,-114.379,-24.082,21.592,-43.531
C06645=1014.722,-49.578,-114.347,-24.081,21.592,-43.536
C06646=1014.721,-49.975,-114.316,-24.080,21.593,-43.542
C06647=1014.718,-50.372,-114.284,-24.080,21.594,-43.547
C06648=1014.715,-50.769,-114.252,-24.079,21.595,-43.553
C06649=1014.713,-51.166,-114.221,-24.078,21.595,-43.558
C06650=1014.710,-51.563,-114.189,-24.077,21.596,-43.564
C06651=1014.707,-51.961,-114.158,-24.077,21.597,-43.570
C06652=1014.705,-52.357,-114.127,-24.076,21.598,-43.575
C06653=1014.702,-52.754,-114.095,-24.075,21.598,-43.581
C06654=1014.700,-53.151,-114.064,-24.074,21.598,-43.588
C06655=1014.698,-53.548,-114.032,-24.073,21.599,-43.593
C06656=1014.695,-53.946,-114.001,-24.073,21.599,-43.599
C06657=1014.692,-54.342,-113.970,-24.072,21.600,-43.604
C06658=1014.689,-54.739,-113.937,-24.071,21.601,-43.610
C06659=1014.686,-55.136,-113.906,-24.071,21.602,-43.616
C06660=1014.684,-55.533,-113.875,-24.070,21.603,-43.621
C06661=1014.681,-55.931,-113.843,-24.069,21.602,-43.627
C06662=1014.678,-56.328,-113.812,-24.068,21.603,-43.632
C06663=1014.675,-56.726,-113.781,-24.067,21.603,-43.639
C06664=1014.672,-57.124,-113.750,-24.067,21.604,-43.645
C06665=1014.669,-57.522,-113.719,-24.066,21.605,-43.651
C06666=1014.666,-57.922,-113.687,-24.065,21.606,-43.656
C06667=1014.663,-58.320,-113.656,-24.064,21.606,-43.662
C06668=1014.660,-58.720,-113.624,-24.064,21.607,-43.667
C06669=1014.658,-59.120,-113.593,-24.063,21.608,-43.673
C06670=1014.654,-59.521,-113.561,-24.062,21.608,-43.680
C06671=1014.651,-59.922,-113.530,-24.061,21.609,-43.686
C06672=1014.647,-60.325,-113.498,-24.061,21.610,-43.691
C06673=1014.645,-60.728,-113.466,-24.060,21.610,-43.697
C06674=1014.642,-61.130,-113.435,-24.059,21.610,-43.702
C06675=1014.638,-61.534,-113.404,-24.058,21.611,-43.708
C06676=1014.635,-61.938,-113.372,-24.057,21.611,-43.715
C06677=1014.632,-62.343,-113.340,-24.057,21.612,-43.720
C06678=1014.628,-62.748,-113.308,-24.056,21.613,-43.726
C06679=1014.625,-63.154,-113.276,-24.055,21.614,-43.732
C06680=1014.621,-63.560,-113.244,-24.054,21.615,-43.737
C06681=1014.618,-63.967,-113.213,-24.053,21.615,-43.744
C06682=1014.614,-64.374,-113.180,-24.053,21.615,-43.750
C06683=1014.610,-64.782,-113.148,-24.052,21.616,-43.756
C06684=1014.607,-65.190,-113.117,-24.051,21.617,-43.761
C06685=1014.603,-65.599,-113.085,-24.050,21.617,-43.768
C06686=1014.600,-66.008,-113.053,-24.049,21.618,-43.774
C06687=1014.595,-66.417,-113.021,-24.049,21.619,-43.780
C06688=1014.592,-66.826,-112.989,-24.048,21.620,-43.785
C06689=1014.588,-67.236,-112.957,-24.047,21.620,-43.791
C06690=1014.584,-67.647,-112.925,-24.046,21.621,-43.798
C06691=1014.581,-68.057,-112.893,-24.046,21.621,-43.804
C06692=1014.577,-68.467,-112.862,-24.045,21.622,-43.809
C06693=1014.572,-68.878,-112.829,-24.044,21.623,-43.815
C06694=1014.569,-69.289,-112.797,-24.043,21.623,-43.822
C06695=1014.564,-69.699,-112.765,-24.042,21.624,-43.827
C06696=1014.560,-70.110,-112.734,-24.042,21.625,-43.833
C06697=1014.556,-70.521,-112.702,-24.041,21.625,-43.839
C06698=1014.552,-70.933,-112.669,-24.040,21.626,-43.846
C06699=1014.548,-71.344,-112.637,-24.039,21.626,-43.851
C06700=1014.544,-71.754,-112.606,-24.039,21.627,-43.857
C06701=1014.540,-72.165,-112.574,-24.038,21.628,-43.865
C06702=1014.535,-72.576,-112.542,-24.037,21.629,-43.870
C06703=1014.531,-72.987,-112.509,-24.036,21.630,-43.876
C06704=1014.527,-73.398,-112.478,-24.035,21.631,-43.881
C06705=1014.523,-73.809,-112.446,-24.034,21.631,-43.888
C06706=1014.517,-74.220,-112.414,-24.034,21.632,-43.894
C06707=1014.513,-74.630,-112.383,-24.033,21.632,-43.900
C06708=1014.508,-75.040,-112.351,-24.032,21.633,-43.905
C06709=1014.504,-75.450,-112.319,-24.031,21.633,-43.912
C06710=1014.500,-75.861,-112.288,-24.031,21.634,-43.918
C06711=1014.495,-76.270,-112.256,-24.030,21.635,-43.924
C06712=1014.490,-76.680,-112.224,-24.029,21.636,-43.929
C06713=1014.485,-77.089,-112.192,-24.028,21.636,-43.936
C06714=1014.481,-77.497,-112.160,-24.027,21.637,-43.942
C06715=1014.476,-77.906,-112.129,-24.027,21.637,-43.948
C06716=1014.471,-78.314,-112.098,-24.026,21.638,-43.953
C06717=1014.467,-78.722,-112.066,-24.025,21.638,-43.960
C06718=1014.461,-79.129,-112.035,-24.024,21.639,-43.966
C06719=1014.457,-79.536,-112.003,-24.023,21.640,-43.972
C06720=1014.451,-79.942,-111.972,-24.023,21.641,-43.977
C06721=1014.446,-80.348,-111.941,-24.022,21.641,-43.984
C06722=1014.441,-80.753,-111.909,-24.021,21.642,-43.990
C06723=1014.436,-81.157,-111.878,-24.020,21.643,-43.995
C06724=1014.432,-81.562,-111.847,-24.020,21.643,-44.001
C06725=1014.426,-81.965,-111.816,-24.019,21.644,-44.007
C06726=1014.421,-82.368,-111.785,-24.018,21.644,-44.014
C06727=1014.416,-82.770,-111.754,-24.017,21.645,-44.019
C06728=1014.411,-83.172,-111.723,-24.016,21.646,-44.025
C06729=1014.406,-83.573,-111.692,-24.016,21.647,-44.031
C06730=1014.401,-83.973,-111.662,-24.015,21.648,-44.036
C06731=1014.395,-84.373,-111.631,-24.014,21.648,-44.043
C06732=1014.390,-84.779,-111.600,-24.013,21.649,-44.049
C06733=1014.386,-85.003,-111.582,-24.013,21.649,-44.053
C06734=1014.383,-85.244,-111.564,-24.012,21.650,-44.056
C06735=1014.379,-85.498,-111.544,-24.012,21.649,-44.060
C06736=1014.376,-85.752,-111.525,-24.012,21.650,-44.062
C06737=1014.373,-85.999,-111.505,-24.011,21.650,-44.065
C06738=1014.370,-86.228,-111.489,-24.011,21.651,-44.069
C06739=1014.364,-86.638,-111.456,-24.010,21.652,-44.077
C06740=1014.359,-87.026,-111.427,-24.009,21.652,-44.082
C06741=1014.353,-87.406,-111.399,-24.008,21.652,-44.087
C06742=1014.348,-87.778,-111.369,-24.007,21.653,-44.093
C06743=1014.343,-88.151,-111.341,-24.007,21.654,-44.099
C06744=1014.337,-88.526,-111.312,-24.006,21.655,-44.104
C06745=1014.331,-88.934,-111.281,-24.005,21.656,-44.112
C06746=1014.328,-89.181,-111.262,-24.005,21.656,-44.116
C06747=1014.324,-89.455,-111.241,-24.004,21.657,-44.117
C06748=1014.320,-89.740,-111.219,-24.004,21.656,-44.121
C06749=1014.315,-90.015,-111.198,-24.003,21.657,-44.124
C06750=1014.311,-90.265,-111.178,-24.003,21.657,-44.128
C06751=1014.309,-90.483,-111.162,-24.002,21.658,-44.132
C06752=1014.302,-90.879,-111.131,-24.002,21.659,-44.138
C06753=1014.296,-91.274,-111.101,-24.001,21.659,-44.145
C06754=1014.291,-91.666,-111.071,-24.000,21.660,-44.150
C06755=1014.285,-92.059,-111.041,-23.999,21.660,-44.156
C06756=1014.279,-92.450,-111.011,-23.999,21.661,-44.162
C06757=1014.273,-92.841,-110.981,-23.998,21.662,-44.167
C06758=1014.266,-93.232,-110.951,-23.997,21.663,-44.173
C06759=1014.260,-93.620,-110.922,-23.996,21.664,-44.178
C06760=1014.254,-94.009,-110.892,-23.996,21.664,-44.184
C06761=1014.247,-94.396,-110.862,-23.995,21.664,-44.189
C06762=1014.241,-94.783,-110.833,-23.994,21.665,-44.195
C06763=1014.234,-95.170,-110.803,-23.994,21.666,-44.200
C06764=1014.228,-95.556,-110.774,-23.993,21.666,-44.207
C06765=1014.221,-95.941,-110.744,-23.992,21.667,-44.213
C06766=1014.216,-96.326,-110.715,-23.991,21.668,-44.219
C06767=1014.210,-96.710,-110.685,-23.990,21.668,-44.224
C06768=1014.203,-97.094,-110.655,-23.990,21.669,-44.230
C06769=1014.196,-97.477,-110.626,-23.989,21.669,-44.235
C06770=1014.190,-97.861,-110.597,-23.988,21.670,-44.241
C06771=1014.183,-98.244,-110.567,-23.988,21.671,-44.246
C06772=1014.176,-98.628,-110.538,-23.987,21.672,-44.252
C06773=1014.170,-99.011,-110.509,-23.986,21.673,-44.258
C06774=1014.163,-99.394,-110.480,-23.985,21.673,-44.263
C06775=1014.156,-99.779,-110.451,-23.985,21.673,-44.268
C06776=1014.149,-100.163,-110.421,-23.984,21.674,-44.274
C06777=1014.143,-100.547,-110.391,-23.983,21.675,-44.280
C06778=1014.135,-100.934,-110.362,-23.982,21.676,-44.285
C06779=1014.129,-101.319,-110.333,-23.982,21.677,-44.291
C06780=1014.121,-101.706,-110.303,-23.981,21.676,-44.296
C06781=1014.115,-102.093,-110.274,-23.980,21.677,-44.302
C06782=1014.106,-102.481,-110.244,-23.980,21.678,-44.307
C06783=1014.099,-102.870,-110.214,-23.979,21.678,-44.314
C06784=1014.092,-103.259,-110.185,-23.978,21.679,-44.320
C06785=1014.085,-103.649,-110.155,-23.977,21.680,-44.326
C06786=1014.078,-104.039,-110.125,-23.976,21.681,-44.331
C06787=1014.070,-104.430,-110.095,-23.976,21.682,-44.337
C06788=1014.062,-104.822,-110.065,-23.975,21.681,-44.342
C06789=1014.054,-105.215,-110.035,-23.974,21.682,-44.348
C06790=1014.046,-105.607,-110.005,-23.974,21.683,-44.353
C06791=1014.038,-106.000,-109.975,-23.973,21.684,-44.359
C06792=1014.031,-106.393,-109.945,-23.972,21.685,-44.365
C06793=1014.023,-106.786,-109.915,-23.971,21.686,-44.370
C06794=1014.015,-107.180,-109.885,-23.971,21.686,-44.376
C06795=1014.007,-107.572,-109.855,-23.970,21.687,-44.383
C06796=1013.999,-107.966,-109.825,-23.969,21.687,-44.388
C06797=1013.991,-108.359,-109.795,-23.968,21.688,-44.394
C06798=1013.982,-108.752,-109.764,-23.968,21.688,-44.399
C06799=1013.975,-109.145,-109.734,-23.967,21.689,-44.405
C06800=1013.966,-109.538,-109.704,-23.966,21.690,-44.411
C06801=1013.958,-109.931,-109.674,-23.965,21.691,-44.416
C06802=1013.949,-110.325,-109.644,-23.965,21.691,-44.422
C06803=1013.940,-110.717,-109.614,-23.964,21.692,-44.427
C06804=1013.932,-111.110,-109.583,-23.963,21.693,-44.433
C06805=1013.924,-111.503,-109.554,-23.963,21.694,-44.439
C06806=1013.920,-111.672,-109.540,-23.962,21.693,-44.442
C06807=1013.893,-112.900,-109.447,-24.170,22.413,-43.999
C06808=1013.887,-113.130,-109.428,-24.208,22.550,-43.917
C06809=1013.882,-113.361,-109.411,-24.246,22.687,-43.835
C06810=1013.876,-113.593,-109.393,-24.285,22.824,-43.752
C06811=1013.872,-113.825,-109.376,-24.323,22.962,-43.671
C06812=1013.867,-114.056,-109.358,-24.361,23.100,-43.589
C06813=1013.862,-114.287,-109.340,-24.399,23.238,-43.508
C06814=1013.856,-114.518,-109.322,-24.437,23.378,-43.427
C06815=1013.851,-114.750,-109.304,-24.474,23.517,-43.345
C06816=1013.846,-114.981,-109.287,-24.512,23.656,-43.264
C06817=1013.841,-115.212,-109.269,-24.549,23.797,-43.183
C06818=1013.835,-115.444,-109.250,-24.586,23.936,-43.102
C06819=1013.830,-115.675,-109.233,-24.623,24.078,-43.023
C06820=1013.825,-115.906,-109.215,-24.660,24.218,-42.942
C06821=1013.820,-116.136,-109.197,-24.697,24.359,-42.863
C06822=1013.815,-116.369,-109.179,-24.733,24.501,-42.783
C06823=1013.809,-116.599,-109.162,-24.770,24.643,-42.704
C06824=1013.804,-116.831,-109.144,-24.806,24.786,-42.624
C06825=1013.799,-117.061,-109.126,-24.842,24.928,-42.546
C06826=1013.794,-117.293,-109.108,-24.878,25.072,-42.468
C06827=1013.789,-117.524,-109.089,-24.914,25.215,-42.388
C06828=1013.783,-117.755,-109.072,-24.950,25.359,-42.311
C06829=1013.778,-117.986,-109.054,-24.986,25.504,-42.232
C06830=1013.772,-118.218,-109.036,-25.021,25.649,-42.154
C06831=1013.768,-118.449,-109.018,-25.057,25.793,-42.077
C06832=1013.762,-118.680,-109.001,-25.092,25.938,-41.999
C06833=1013.757,-118.911,-108.982,-25.127,26.083,-41.922
C06834=1013.752,-119.143,-108.964,-25.162,26.230,-41.845
C06835=1013.746,-119.373,-108.946,-25.196,26.376,-41.768
C06836=1013.742,-119.605,-108.928,-25.231,26.522,-41.691
C06837=1013.736,-119.835,-108.910,-25.266,26.670,-41.615
C06838=1013.730,-120.067,-108.892,-25.300,26.817,-41.539
C06839=1013.725,-120.298,-108.874,-25.334,26.965,-41.464
C06840=1013.720,-120.529,-108.856,-25.368,27.113,-41.388
C06841=1013.715,-120.760,-108.838,-25.402,27.260,-41.313
C06842=1013.708,-121.045,-108.816,-25.443,27.444,-41.220
C06843=1013.699,-121.453,-108.784,-25.503,27.708,-41.087
C06844=1013.694,-121.685,-108.766,-25.536,27.858,-41.013
C06845=1013.688,-121.916,-108.748,-25.569,28.009,-40.939
C06846=1013.683,-122.147,-108.730,-25.602,28.159,-40.865
C06847=1013.678,-122.377,-108.712,-25.635,28.309,-40.791
C06848=1013.672,-122.609,-108.694,-25.668,28.460,-40.718
C06849=1013.666,-122.840,-108.676,-25.700,28.611,-40.645
C06850=1013.662,-123.071,-108.658,-25.733,28.763,-40.571
C06851=1013.657,-123.302,-108.640,-25.765,28.915,-40.498
C06852=1013.651,-123.533,-108.621,-25.797,29.067,-40.425
C06853=1013.646,-123.764,-108.603,-25.829,29.220,-40.355
C06854=1013.641,-123.995,-108.585,-25.861,29.373,-40.283
C06855=1013.635,-124.225,-108.567,-25.893,29.526,-40.211
C06856=1013.630,-124.457,-108.549,-25.925,29.680,-40.139
C06857=1013.625,-124.688,-108.530,-25.956,29.834,-40.067
C06858=1013.619,-124.919,-108.512,-25.987,29.988,-39.996
C06859=1013.615,-125.150,-108.494,-26.019,30.143,-39.925
C06860=1013.608,-125.381,-108.476,-26.050,30.298,-39.855
C06861=1013.603,-125.612,-108.458,-26.081,30.453,-39.784
C06862=1013.598,-125.842,-108.439,-26.111,30.609,-39.714
C06863=1013.593,-126.074,-108.422,-26.142,30.764,-39.645
C06864=1013.587,-126.305,-108.403,-26.172,30.921,-39.574
C06865=1013.582,-126.536,-108.384,-26.203,31.077,-39.506
C06866=1013.577,-126.766,-108.366,-26.233,31.235,-39.436
C06867=1013.572,-126.997,-108.349,-26.263,31.392,-39.367
C06868=1013.566,-127.229,-108.330,-26.293,31.549,-39.299
C06869=1013.561,-127.459,-108.312,-26.323,31.707,-39.231
C06870=1013.556,-127.690,-108.293,-26.352,31.865,-39.162
C06871=1013.550,-127.921,-108.275,-26.382,32.022,-39.095
C06872=1013.545,-128.153,-108.257,-26.411,32.181,-39.027
C06873=1013.540,-128.384,-108.239,-26.440,32.341,-38.960
C06874=1013.535,-128.614,-108.220,-26.469,32.500,-38.893
C06875=1013.529,-128.845,-108.202,-26.498,32.660,-38.826
C06876=1013.523,-129.076,-108.184,-26.527,32.820,-38.760
C06877=1013.517,-129.351,-108.162,-26.561,33.010,-38.680
C06878=1013.508,-129.769,-108.129,-26.613,33.302,-38.561
C06879=1013.503,-130.000,-108.110,-26.641,33.462,-38.495
C06880=1013.497,-130.231,-108.092,-26.669,33.623,-38.430
C06881=1013.492,-130.461,-108.073,-26.697,33.786,-38.365
C06882=1013.487,-130.692,-108.055,-26.725,33.948,-38.301
C06883=1013.481,-130.923,-108.036,-26.753,34.110,-38.237
C06884=1013.476,-131.154,-108.018,-26.780,34.273,-38.171
C06885=1013.471,-131.385,-107.999,-26.808,34.435,-38.108
C06886=1013.466,-131.615,-107.981,-26.835,34.598,-38.044
C06887=1013.460,-131.847,-107.962,-26.862,34.761,-37.981
C06888=1013.456,-132.078,-107.945,-26.889,34.925,-37.917
C06889=1013.450,-132.309,-107.926,-26.917,35.090,-37.854
C06890=1013.445,-132.539,-107.908,-26.943,35.253,-37.792
C06891=1013.440,-132.771,-107.889,-26.970,35.418,-37.730
C06892=1013.434,-133.002,-107.871,-26.996,35.582,-37.669
C06893=1013.429,-133.232,-107.852,-27.023,35.747,-37.607
C06894=1013.424,-133.463,-107.834,-27.049,35.912,-37.545
C06895=1013.419,-133.694,-107.815,-27.075,36.076,-37.484
C06896=1013.413,-133.925,-107.797,-27.101,36.242,-37.423
C06897=1013.408,-134.156,-107.778,-27.127,36.408,-37.362
C06898=1013.834,-134.175,-108.121,-24.568,24.003,-43.339
C06899=1013.841,-133.944,-108.140,-24.522,23.831,-43.439
C06900=1013.848,-133.714,-108.157,-24.475,23.659,-43.540
C06901=1013.854,-133.483,-108.174,-24.429,23.487,-43.642
C06902=1013.860,-133.252,-108.192,-24.382,23.316,-43.742
C06903=1013.867,-133.021,-108.210,-24.334,23.145,-43.845
C06904=1013.873,-132.790,-108.228,-24.287,22.975,-43.948
C06905=1013.879,-132.559,-108.245,-24.239,22.804,-44.051
C06906=1013.886,-132.329,-108.262,-24.190,22.634,-44.155
C06907=1013.920,-131.102,-108.356,-23.926,21.727,-44.719
C06908=1013.930,-130.698,-108.387,-23.927,21.727,-44.714
C06909=1013.942,-130.307,-108.417,-23.928,21.726,-44.708
C06910=1013.952,-129.914,-108.447,-23.929,21.725,-44.703
C06911=1013.962,-129.522,-108.477,-23.929,21.724,-44.697
C06912=1013.973,-129.130,-108.506,-23.930,21.723,-44.691
C06913=1013.984,-128.738,-108.536,-23.931,21.723,-44.686
C06914=1013.994,-128.346,-108.566,-23.932,21.723,-44.680
C06915=1014.004,-127.953,-108.595,-23.932,21.722,-44.675
C06916=1014.014,-127.562,-108.625,-23.933,21.721,-44.669
C06917=1014.024,-127.169,-108.655,-23.934,21.720,-44.664
C06918=1014.034,-126.777,-108.684,-23.934,21.719,-44.658
C06919=1014.045,-126.384,-108.714,-23.935,21.719,-44.652
C06920=1014.055,-125.992,-108.744,-23.936,21.719,-44.647
C06921=1014.065,-125.601,-108.773,-23.936,21.718,-44.642
C06922=1014.075,-125.209,-108.803,-23.937,21.717,-44.636
C06923=1014.084,-124.816,-108.833,-23.938,21.716,-44.630
C06924=1014.094,-124.424,-108.862,-23.939,21.715,-44.625
C06925=1014.104,-124.031,-108.892,-23.939,21.714,-44.619
C06926=1014.113,-123.639,-108.922,-23.940,21.715,-44.614
C06927=1014.123,-123.247,-108.951,-23.941,21.714,-44.608
C06928=1014.132,-122.855,-108.981,-23.941,21.713,-44.603
C06929=1014.142,-122.462,-109.011,-23.942,21.712,-44.597
C06930=1014.151,-122.070,-109.041,-23.943,21.711,-44.591
C06931=1014.160,-121.678,-109.070,-23.943,21.710,-44.586
C06932=1014.170,-121.286,-109.100,-23.944,21.710,-44.580
C06933=1014.179,-120.892,-109.129,-23.945,21.710,-44.575
C06934=1014.187,-120.500,-109.159,-23.946,21.709,-44.569
C06935=1014.196,-120.108,-109.189,-23.946,21.708,-44.564
C06936=1014.205,-119.715,-109.218,-23.947,21.707,-44.558
C06937=1014.215,-119.323,-109.247,-23.948,21.706,-44.553
C06938=1014.223,-118.931,-109.277,-23.948,21.706,-44.547
C06939=1014.232,-118.538,-109.306,-23.949,21.705,-44.541
C06940=1014.240,-118.146,-109.337,-23.950,21.705,-44.536
C06941=1014.249,-117.753,-109.366,-23.951,21.705,-44.529
C06942=1014.258,-117.361,-109.396,-23.952,21.704,-44.523
C06943=1014.266,-116.968,-109.425,-23.952,21.703,-44.518
C06944=1014.276,-116.575,-109.455,-23.953,21.702,-44.512
C06945=1014.283,-116.183,-109.484,-23.954,21.701,-44.507
C06946=1014.292,-115.791,-109.514,-23.954,21.700,-44.501
C06947=1014.301,-115.398,-109.543,-23.955,21.701,-44.496
C06948=1014.308,-115.005,-109.573,-23.956,21.700,-44.490
C06949=1014.317,-114.613,-109.603,-23.957,21.699,-44.485
C06950=1014.325,-114.220,-109.632,-23.957,21.698,-44.479
C06951=1014.334,-113.827,-109.661,-23.958,21.697,-44.473
C06952=1014.341,-113.434,-109.691,-23.959,21.696,-44.468
C06953=1014.349,-113.041,-109.721,-23.959,21.696,-44.462
C06954=1014.357,-112.649,-109.750,-23.960,21.695,-44.456
C06955=1014.365,-112.256,-109.780,-23.961,21.694,-44.451
C06956=1014.373,-111.863,-109.810,-23.962,21.694,-44.446
C06957=1014.381,-111.470,-109.839,-23.963,21.694,-44.439
C06958=1014.388,-111.077,-109.869,-23.963,21.693,-44.433
C06959=1014.396,-110.684,-109.899,-23.964,21.692,-44.427
C06960=1014.404,-110.291,-109.928,-23.965,21.691,-44.422
C06961=1014.411,-109.899,-109.958,-23.965,21.691,-44.416
C06962=1014.419,-109.506,-109.987,-23.966,21.690,-44.411
C06963=1014.426,-109.112,-110.016,-23.967,21.689,-44.405
C06964=1014.434,-108.719,-110.046,-23.968,21.688,-44.399
C06965=1014.442,-108.326,-110.076,-23.968,21.688,-44.394
C06966=1014.450,-107.933,-110.105,-23.969,21.687,-44.388
C06967=1014.456,-107.540,-110.135,-23.970,21.687,-44.383
C06968=1014.464,-107.147,-110.164,-23.971,21.686,-44.376
C06969=1014.471,-106.753,-110.194,-23.971,21.686,-44.370
C06970=1014.478,-106.361,-110.224,-23.972,21.685,-44.365
C06971=1014.486,-105.968,-110.253,-23.973,21.684,-44.359
C06972=1014.492,-105.575,-110.283,-23.974,21.683,-44.353
C06973=1014.499,-105.182,-110.312,-23.974,21.682,-44.348
C06974=1014.507,-104.790,-110.342,-23.975,21.681,-44.342
C06975=1014.513,-104.399,-110.371,-23.976,21.682,-44.337
C06976=1014.520,-104.007,-110.401,-23.976,21.681,-44.331
C06977=1014.527,-103.617,-110.430,-23.977,21.680,-44.326
C06978=1014.533,-103.227,-110.460,-23.978,21.679,-44.320
C06979=1014.540,-102.837,-110.489,-23.979,21.678,-44.314
C06980=1014.547,-102.449,-110.518,-23.980,21.678,-44.307
C06981=1014.553,-102.061,-110.548,-23.980,21.677,-44.302
C06982=1014.560,-101.674,-110.577,-23.981,21.676,-44.296
C06983=1014.566,-101.287,-110.606,-23.982,21.677,-44.291
C06984=1014.573,-100.902,-110.635,-23.982,21.676,-44.285
C06985=1014.580,-100.516,-110.664,-23.983,21.675,-44.280
C06986=1014.585,-100.131,-110.693,-23.984,21.674,-44.274
C06987=1014.592,-99.747,-110.722,-23.985,21.673,-44.268
C06988=1014.598,-99.363,-110.751,-23.985,21.673,-44.263
C06989=1014.604,-98.979,-110.780,-23.986,21.673,-44.258
C06990=1014.610,-98.596,-110.809,-23.987,21.672,-44.252
C06991=1014.616,-98.213,-110.838,-23.988,21.671,-44.246
C06992=1014.623,-97.830,-110.866,-23.988,21.670,-44.241
C06993=1014.628,-97.446,-110.895,-23.989,21.669,-44.235
C06994=1014.635,-97.062,-110.925,-23.990,21.669,-44.230
C06995=1014.641,-96.679,-110.954,-23.990,21.668,-44.224
C06996=1014.646,-96.294,-110.984,-23.991,21.668,-44.219
C06997=1014.653,-95.910,-111.012,-23.992,21.667,-44.213
C06998=1014.658,-95.525,-111.042,-23.993,21.666,-44.207
C06999=1014.664,-95.139,-111.070,-23.994,21.666,-44.200
C07000=1014.670,-94.753,-111.100,-23.994,21.665,-44.195
C07001=1014.675,-94.366,-111.129,-23.995,21.664,-44.189
C07002=1014.682,-93.978,-111.158,-23.996,21.664,-44.184
C07003=1014.687,-93.590,-111.187,-23.996,21.664,-44.178
C07004=1014.692,-93.201,-111.217,-23.997,21.663,-44.173
C07005=1014.698,-92.811,-111.247,-23.998,21.662,-44.167
C07006=1014.704,-92.420,-111.277,-23.999,21.661,-44.162
C07007=1014.710,-92.028,-111.306,-23.999,21.660,-44.156
C07008=1014.715,-91.636,-111.336,-24.000,21.660,-44.150
C07009=1014.721,-91.243,-111.365,-24.001,21.659,-44.145
C07010=1014.726,-90.849,-111.395,-24.002,21.659,-44.138
C07011=1014.732,-90.453,-111.426,-24.002,21.658,-44.132
C07012=1014.734,-90.234,-111.442,-24.003,21.657,-44.128
C07013=1014.738,-89.984,-111.461,-24.003,21.657,-44.124
C07014=1014.742,-89.709,-111.482,-24.004,21.656,-44.121
C07015=1014.746,-89.424,-111.504,-24.004,21.657,-44.117
C07016=1014.750,-89.150,-111.525,-24.005,21.656,-44.116
C07017=1014.753,-88.903,-111.543,-24.005,21.656,-44.112
C07018=1014.758,-88.496,-111.574,-24.006,21.655,-44.104
C07019=1014.763,-88.120,-111.602,-24.007,21.654,-44.099
C07020=1014.768,-87.748,-111.631,-24.007,21.653,-44.093
C07021=1014.773,-87.375,-111.660,-24.008,21.652,-44.087
C07022=1014.778,-86.996,-111.688,-24.009,21.652,-44.082
C07023=1014.783,-86.608,-111.718,-24.010,21.652,-44.077
C07024=1014.788,-86.199,-111.749,-24.011,21.651,-44.069
C07025=1014.791,-85.968,-111.766,-24.011,21.650,-44.065
C07026=1014.794,-85.722,-111.785,-24.012,21.650,-44.062
C07027=1014.798,-85.467,-111.805,-24.012,21.649,-44.060
C07028=1014.801,-85.214,-111.824,-24.012,21.650,-44.056
C07029=1014.804,-84.973,-111.843,-24.013,21.649,-44.053
C07030=1014.806,-84.749,-111.859,-24.013,21.649,-44.049
C07031=1014.811,-84.343,-111.891,-24.014,21.648,-44.043
C07032=1014.816,-83.944,-111.921,-24.015,21.648,-44.036
C07033=1014.821,-83.543,-111.952,-24.016,21.647,-44.031
C07034=1014.826,-83.142,-111.982,-24.016,21.646,-44.025
C07035=1014.831,-82.740,-112.013,-24.017,21.645,-44.019
C07036=1014.835,-82.338,-112.043,-24.018,21.644,-44.014
C07037=1014.840,-81.936,-112.074,-24.019,21.644,-44.007
C07038=1014.846,-81.531,-112.105,-24.020,21.643,-44.001
C07039=1014.849,-81.128,-112.136,-24.020,21.643,-43.995
C07040=1014.855,-80.724,-112.167,-24.021,21.642,-43.990
C07041=1014.859,-80.318,-112.198,-24.022,21.641,-43.984
C07042=1014.863,-79.912,-112.229,-24.023,21.641,-43.977
C07043=1014.868,-79.506,-112.260,-24.023,21.640,-43.972
C07044=1014.873,-79.099,-112.292,-24.024,21.639,-43.966
C07045=1014.878,-78.692,-112.323,-24.025,21.638,-43.960
C07046=1014.882,-78.285,-112.354,-24.026,21.638,-43.953
C07047=1014.887,-77.876,-112.385,-24.027,21.637,-43.948
C07048=1014.891,-77.468,-112.417,-24.027,21.637,-43.942
C07049=1014.896,-77.059,-112.448,-24.028,21.636,-43.936
C07050=1014.899,-76.650,-112.479,-24.029,21.636,-43.929
C07051=1014.904,-76.240,-112.511,-24.030,21.635,-43.924
C07052=1014.908,-75.831,-112.542,-24.031,21.634,-43.918
C07053=1014.912,-75.421,-112.574,-24.031,21.633,-43.912
C07054=1014.916,-75.011,-112.605,-24.032,21.633,-43.905
C07055=1014.921,-74.601,-112.637,-24.033,21.632,-43.900
C07056=1014.926,-74.190,-112.669,-24.034,21.632,-43.894
C07057=1014.929,-73.779,-112.700,-24.034,21.631,-43.888
C07058=1014.933,-73.369,-112.731,-24.035,21.631,-43.881
C07059=1014.937,-72.957,-112.763,-24.036,21.630,-43.876
C07060=1014.942,-72.548,-112.795,-24.037,21.629,-43.870
C07061=1014.946,-72.136,-112.827,-24.038,21.628,-43.865
C07062=1014.949,-71.725,-112.859,-24.039,21.627,-43.857
C07063=1014.954,-71.314,-112.890,-24.039,21.626,-43.851
C07064=1014.957,-70.904,-112.922,-24.040,21.626,-43.846
C07065=1014.961,-70.492,-112.954,-24.041,21.625,-43.839
C07066=1014.965,-70.081,-112.986,-24.042,21.625,-43.833
C07067=1014.969,-69.670,-113.018,-24.042,21.624,-43.827
C07068=1014.972,-69.259,-113.049,-24.043,21.623,-43.822
C07069=1014.976,-68.849,-113.081,-24.044,21.623,-43.815
C07070=1014.980,-68.437,-113.113,-24.045,21.622,-43.809
C07071=1014.984,-68.027,-113.145,-24.046,21.621,-43.804
C07072=1014.987,-67.617,-113.176,-24.046,21.621,-43.798
C07073=1014.991,-67.207,-113.209,-24.047,21.620,-43.791
C07074=1014.994,-66.797,-113.239,-24.048,21.620,-43.785
C07075=1014.998,-66.387,-113.272,-24.049,21.619,-43.780
C07076=1015.002,-65.978,-113.303,-24.049,21.618,-43.774
C07077=1015.004,-65.570,-113.335,-24.050,21.617,-43.768
C07078=1015.009,-65.161,-113.367,-24.051,21.617,-43.761
C07079=1015.012,-64.753,-113.399,-24.052,21.616,-43.756
C07080=1015.015,-64.345,-113.431,-24.053,21.615,-43.750
C07081=1015.018,-63.938,-113.463,-24.053,21.615,-43.744
C07082=1015.022,-63.531,-113.494,-24.054,21.615,-43.737
C07083=1015.025,-63.125,-113.526,-24.055,21.614,-43.732
C07084=1015.028,-62.719,-113.558,-24.056,21.613,-43.726
C07085=1015.032,-62.314,-113.589,-24.057,21.612,-43.720
C07086=1015.035,-61.910,-113.621,-24.057,21.611,-43.715
C07087=1015.037,-61.505,-113.653,-24.058,21.611,-43.708
C07088=1015.041,-61.102,-113.684,-24.059,21.610,-43.702
C07089=1015.044,-60.698,-113.715,-24.060,21.610,-43.697
C07090=1015.046,-60.296,-113.747,-24.061,21.610,-43.691
C07091=1015.049,-59.894,-113.778,-24.061,21.609,-43.686
C07092=1015.053,-59.493,-113.809,-24.062,21.608,-43.680
C07093=1015.055,-59.092,-113.841,-24.063,21.608,-43.673
C07094=1015.059,-58.692,-113.872,-24.064,21.607,-43.667
C07095=1015.061,-58.291,-113.903,-24.064,21.606,-43.662
C07096=1015.064,-57.892,-113.935,-24.065,21.606,-43.656
C07097=1015.067,-57.494,-113.966,-24.066,21.605,-43.651
C07098=1015.069,-57.095,-113.998,-24.067,21.604,-43.645
C07099=1015.072,-56.697,-114.029,-24.067,21.603,-43.639
C07100=1015.075,-56.299,-114.060,-24.068,21.603,-43.632
C07101=1015.078,-55.902,-114.091,-24.069,21.602,-43.627
C07102=1015.080,-55.505,-114.122,-24.070,21.603,-43.621
C07103=1015.083,-55.107,-114.154,-24.071,21.602,-43.616
C07104=1015.085,-54.710,-114.185,-24.071,21.601,-43.610
C07105=1015.088,-54.313,-114.217,-24.072,21.600,-43.604
C07106=1015.090,-53.916,-114.248,-24.073,21.599,-43.599
C07107=1015.093,-53.519,-114.279,-24.073,21.599,-43.593
C07108=1015.095,-53.123,-114.310,-24.074,21.598,-43.588
C07109=1015.098,-52.725,-114.341,-24.075,21.598,-43.581
C07110=1015.100,-52.329,-114.372,-24.076,21.598,-43.575
C07111=1015.102,-51.932,-114.405,-24.077,21.597,-43.570
C07112=1015.105,-51.535,-114.436,-24.077,21.596,-43.564
C07113=1015.108,-51.138,-114.467,-24.078,21.595,-43.558
C07114=1015.110,-50.741,-114.498,-24.079,21.595,-43.553
C07115=1015.112,-50.343,-114.530,-24.080,21.594,-43.547
C07116=1015.114,-49.947,-114.561,-24.080,21.593,-43.542
C07117=1015.116,-49.549,-114.593,-24.081,21.592,-43.536
C07118=1015.119,-49.153,-114.624,-24.082,21.592,-43.531
C07119=1015.121,-48.755,-114.656,-24.083,21.592,-43.525
C07120=1015.123,-48.358,-114.687,-24.084,21.592,-43.518
C07121=1015.125,-47.961,-114.719,-24.084,21.591,-43.512
C07122=1015.127,-47.564,-114.751,-24.085,21.590,-43.507
C07123=1015.129,-47.166,-114.782,-24.086,21.589,-43.501
C07124=1015.131,-46.770,-114.814,-24.086,21.588,-43.496
C07125=1015.133,-46.372,-114.846,-24.087,21.589,-43.490
C07126=1015.135,-45.975,-114.877,-24.088,21.588,-43.485
C07127=1015.137,-45.578,-114.909,-24.089,21.587,-43.479
C07128=1015.139,-45.181,-114.940,-24.089,21.586,-43.473
C07129=1015.140,-44.784,-114.972,-24.090,21.585,-43.468
C07130=1015.142,-44.386,-115.004,-24.091,21.585,-43.462
C07131=1015.144,-43.989,-115.035,-24.092,21.585,-43.457
C07132=1015.146,-43.592,-115.067,-24.092,21.584,-43.451
C07133=1015.148,-43.195,-115.098,-24.093,21.584,-43.444
C07134=1015.150,-42.797,-115.130,-24.094,21.583,-43.439
C07135=1015.151,-42.400,-115.162,-24.095,21.582,-43.433
C07136=1015.153,-42.002,-115.194,-24.096,21.582,-43.427
C07137=1015.155,-41.606,-115.226,-24.096,21.582,-43.422
C07138=1015.157,-41.208,-115.258,-24.097,21.581,-43.417
C07139=1015.158,-40.811,-115.289,-24.098,21.580,-43.411
C07140=1015.161,-40.413,-115.321,-24.099,21.579,-43.405
C07141=1015.162,-40.016,-115.353,-24.099,21.579,-43.400
C07142=1015.163,-39.619,-115.385,-24.100,21.578,-43.394
C07143=1015.165,-39.222,-115.417,-24.101,21.578,-43.389
C07144=1015.166,-38.825,-115.449,-24.102,21.577,-43.383
C07145=1015.168,-38.427,-115.481,-24.102,21.576,-43.378
C07146=1015.169,-38.030,-115.513,-24.103,21.576,-43.372
C07147=1015.171,-37.632,-115.545,-24.104,21.575,-43.366
C07148=1015.172,-37.235,-115.577,-24.105,21.575,-43.361
C07149=1015.174,-36.838,-115.609,-24.105,21.574,-43.356
C07150=1015.175,-36.440,-115.641,-24.106,21.573,-43.350
C07151=1015.177,-36.043,-115.673,-24.107,21.573,-43.344
C07152=1015.178,-35.645,-115.705,-24.107,21.572,-43.339
C07153=1015.180,-35.248,-115.737,-24.108,21.572,-43.334
C07154=1015.180,-34.851,-115.769,-24.109,21.571,-43.328
C07155=1015.182,-34.453,-115.802,-24.110,21.571,-43.321
C07156=1015.183,-34.056,-115.833,-24.111,21.570,-43.315
C07157=1015.185,-33.658,-115.866,-24.111,21.570,-43.310
C07158=1015.185,-33.261,-115.898,-24.112,21.570,-43.304
C07159=1015.187,-32.864,-115.929,-24.113,21.569,-43.299
C07160=1015.188,-32.466,-115.962,-24.114,21.568,-43.293
C07161=1015.189,-32.069,-115.994,-24.114,21.567,-43.287
C07162=1015.190,-31.671,-116.026,-24.115,21.568,-43.282
